C05471=1216.995,158.633,-53.196,-177.937,5.940,148.445
C05472=1217.000,158.384,-53.175,-177.940,5.938,148.445
C05473=1217.005,158.135,-53.154,-177.943,5.937,148.446
C05474=1217.009,157.886,-53.131,-177.945,5.936,148.446
C05475=1217.014,157.637,-53.110,-177.947,5.934,148.446
C05476=1217.019,157.388,-53.089,-177.950,5.933,148.447
C05477=1217.023,157.139,-53.067,-177.953,5.931,148.447
C05478=1217.028,156.890,-53.046,-177.955,5.930,148.448
C05479=1217.033,156.641,-53.025,-177.958,5.929,148.448
C05480=1217.038,156.393,-53.003,-177.961,5.927,148.449
C05481=1217.042,156.143,-52.982,-177.963,5.926,148.449
C05482=1217.047,155.894,-52.960,-177.966,5.925,148.450
C05483=1217.052,155.645,-52.938,-177.968,5.923,148.450
C05484=1217.056,155.396,-52.918,-177.971,5.922,148.451
C05485=1217.061,155.147,-52.896,-177.974,5.920,148.451
C05486=1217.066,154.898,-52.875,-177.976,5.919,148.452
C05487=1217.071,154.649,-52.853,-177.979,5.918,148.452
C05488=1217.075,154.400,-52.831,-177.981,5.917,148.452
C05489=1217.080,154.151,-52.810,-177.984,5.915,148.453
C05490=1217.084,153.902,-52.789,-177.986,5.913,148.453
C05491=1217.089,153.652,-52.768,-177.989,5.912,148.454
C05492=1217.094,153.404,-52.746,-177.992,5.911,148.454
C05493=1217.099,153.154,-52.725,-177.994,5.910,148.455
C05494=1217.104,152.906,-52.704,-177.996,5.908,148.455
C05495=1217.108,152.657,-52.683,-177.999,5.907,148.456
C05496=1217.113,152.407,-52.661,-178.002,5.906,148.456
C05497=1217.118,152.158,-52.640,-178.004,5.905,148.456
C05498=1217.123,151.909,-52.618,-178.007,5.903,148.457
C05499=1217.127,151.661,-52.598,-178.010,5.901,148.457
C05500=1217.131,151.411,-52.576,-178.012,5.900,148.458
C05501=1217.137,151.162,-52.555,-178.015,5.899,148.458
C05502=1217.141,150.913,-52.535,-178.017,5.898,148.459
C05503=1217.146,150.664,-52.513,-178.020,5.896,148.459
C05504=1217.151,150.415,-52.492,-178.022,5.896,148.460
C05505=1217.155,150.166,-52.470,-178.025,5.894,148.460
C05506=1217.160,149.917,-52.450,-178.027,5.893,148.461
C05507=1217.165,149.668,-52.429,-178.030,5.891,148.461
C05508=1217.170,149.419,-52.407,-178.033,5.889,148.462
C05509=1217.174,149.170,-52.387,-178.036,5.889,148.462
C05510=1217.178,148.921,-52.365,-178.038,5.887,148.463
C05511=1217.184,148.671,-52.344,-178.040,5.886,148.463
C05512=1217.188,148.422,-52.323,-178.043,5.885,148.464
C05513=1217.193,148.173,-52.302,-178.046,5.884,148.464
C05514=1217.198,147.925,-52.281,-178.048,5.882,148.464
C05515=1217.203,147.676,-52.260,-178.051,5.881,148.465
C05516=1217.207,147.426,-52.239,-178.053,5.879,148.465
C05517=1217.211,147.177,-52.218,-178.056,5.878,148.466
C05518=1217.216,146.928,-52.197,-178.059,5.877,148.466
C05519=1217.222,146.679,-52.176,-178.061,5.876,148.467
C05520=1217.226,146.430,-52.155,-178.064,5.874,148.467
C05521=1217.231,146.181,-52.134,-178.066,5.874,148.468
C05522=1217.235,145.932,-52.113,-178.069,5.872,148.468
C05523=1217.240,145.682,-52.092,-178.071,5.871,148.469
C05524=1217.245,145.433,-52.071,-178.074,5.869,148.469
C05525=1217.249,145.185,-52.050,-178.076,5.868,148.470
C05526=1217.254,144.935,-52.029,-178.079,5.867,148.470
C05527=1217.259,144.686,-52.009,-178.082,5.865,148.470
C05528=1217.264,144.437,-51.988,-178.084,5.864,148.471
C05529=1217.268,144.188,-51.967,-178.087,5.863,148.471
C05530=1217.274,143.939,-51.946,-178.089,5.862,148.472
C05531=1217.278,143.691,-51.925,-178.093,5.860,148.472
C05532=1217.283,143.441,-51.904,-178.095,5.859,148.473
C05533=1217.287,143.192,-51.884,-178.097,5.857,148.473
C05534=1217.292,142.942,-51.863,-178.100,5.857,148.474
C05535=1217.296,142.694,-51.842,-178.103,5.855,148.474
C05536=1217.302,142.444,-51.821,-178.105,5.854,148.475
C05537=1217.306,142.195,-51.801,-178.108,5.853,148.475
C05538=1217.311,141.946,-51.780,-178.110,5.852,148.476
C05539=1217.316,141.697,-51.760,-178.113,5.850,148.476
C05540=1217.321,141.448,-51.739,-178.115,5.849,148.477
C05541=1217.325,141.199,-51.718,-178.118,5.848,148.477
C05542=1217.330,140.950,-51.697,-178.121,5.847,148.478
C05543=1217.335,140.701,-51.677,-178.123,5.846,148.478
C05544=1217.339,140.452,-51.657,-178.126,5.844,148.479
C05545=1217.344,140.202,-51.636,-178.128,5.843,148.479
C05546=1217.349,139.954,-51.615,-178.131,5.842,148.480
C05547=1217.354,139.704,-51.594,-178.133,5.841,148.480
C05548=1217.359,139.455,-51.574,-178.136,5.839,148.480
C05549=1217.364,139.206,-51.553,-178.138,5.838,148.481
C05550=1217.368,138.957,-51.533,-178.141,5.837,148.482
C05551=1217.373,138.708,-51.512,-178.144,5.836,148.482
C05552=1217.378,138.459,-51.491,-178.146,5.834,148.483
C05553=1217.382,138.210,-51.471,-178.149,5.833,148.483
C05554=1217.387,137.961,-51.450,-178.152,5.832,148.484
C05555=1217.392,137.712,-51.429,-178.154,5.831,148.484
C05556=1217.396,137.463,-51.409,-178.157,5.829,148.485
C05557=1217.401,137.214,-51.388,-178.159,5.828,148.485
C05558=1217.406,136.965,-51.368,-178.162,5.827,148.486
C05559=1217.410,136.716,-51.347,-178.164,5.826,148.486
C05560=1217.416,136.466,-51.327,-178.167,5.824,148.486
C05561=1217.420,136.217,-51.307,-178.170,5.824,148.487
C05562=1217.425,135.968,-51.286,-178.172,5.823,148.487
C05563=1217.429,135.719,-51.266,-178.175,5.821,148.488
C05564=1217.434,135.470,-51.245,-178.177,5.820,148.488
C05565=1217.439,135.221,-51.225,-178.180,5.819,148.489
C05566=1217.443,134.971,-51.205,-178.182,5.818,148.489
C05567=1217.449,134.722,-51.184,-178.185,5.816,148.490
C05568=1217.453,134.473,-51.164,-178.188,5.815,148.490
C05569=1217.457,134.224,-51.143,-178.190,5.814,148.491
C05570=1217.462,133.974,-51.124,-178.193,5.813,148.491
C05571=1217.468,133.706,-51.101,-178.196,5.811,148.492
C05572=1217.473,133.437,-51.080,-178.198,5.810,148.492
C05573=1217.478,133.169,-51.058,-178.201,5.809,148.493
C05574=1217.483,132.900,-51.036,-178.204,5.807,148.493
C05575=1217.488,132.651,-51.016,-178.207,5.807,148.494
C05576=1217.492,132.402,-50.995,-178.209,5.806,148.494
C05577=1217.498,132.153,-50.974,-178.212,5.804,148.495
C05578=1217.502,131.903,-50.955,-178.214,5.803,148.495
C05579=1217.507,131.654,-50.934,-178.217,5.801,148.496
C05580=1217.511,131.406,-50.914,-178.219,5.801,148.497
C05581=1217.517,131.156,-50.894,-178.222,5.799,148.497
C05582=1217.522,130.907,-50.874,-178.225,5.798,148.498
C05583=1217.526,130.658,-50.854,-178.227,5.797,148.498
C05584=1217.531,130.409,-50.834,-178.230,5.796,148.499
C05585=1217.535,130.160,-50.813,-178.232,5.795,148.499
C05586=1217.540,129.910,-50.794,-178.235,5.794,148.500
C05587=1217.545,129.661,-50.773,-178.237,5.793,148.500
C05588=1217.550,129.412,-50.753,-178.240,5.791,148.501
C05589=1217.555,129.163,-50.733,-178.243,5.790,148.501
C05590=1217.559,128.914,-50.713,-178.245,5.790,148.502
C05591=1217.564,128.665,-50.693,-178.248,5.788,148.502
C05592=1217.569,128.416,-50.673,-178.250,5.787,148.503
C05593=1217.573,128.166,-50.653,-178.253,5.785,148.503
C05594=1217.578,127.917,-50.633,-178.255,5.784,148.503
C05595=1217.583,127.668,-50.613,-178.258,5.783,148.504
C05596=1217.588,127.419,-50.592,-178.260,5.782,148.504
C05597=1217.593,127.170,-50.573,-178.263,5.781,148.505
C05598=1217.597,126.921,-50.552,-178.266,5.780,148.505
C05599=1217.602,126.671,-50.533,-178.268,5.779,148.506
C05600=1217.607,126.423,-50.513,-178.271,5.777,148.507
C05601=1217.612,126.173,-50.493,-178.274,5.777,148.507
C05602=1217.616,125.924,-50.473,-178.276,5.776,148.508
C05603=1217.621,125.675,-50.453,-178.279,5.774,148.508
C05604=1217.626,125.426,-50.433,-178.281,5.773,148.509
C05605=1217.631,125.177,-50.413,-178.284,5.772,148.509
C05606=1217.636,124.927,-50.394,-178.286,5.771,148.510
C05607=1217.640,124.678,-50.373,-178.289,5.770,148.510
C05608=1217.645,124.429,-50.354,-178.292,5.768,148.511
C05609=1217.649,124.180,-50.333,-178.294,5.768,148.511
C05610=1217.655,123.931,-50.314,-178.296,5.767,148.512
C05611=1217.659,123.681,-50.294,-178.300,5.765,148.512
C05612=1217.664,123.433,-50.274,-178.302,5.764,148.513
C05613=1217.669,123.183,-50.254,-178.305,5.763,148.513
C05614=1217.674,122.934,-50.235,-178.307,5.762,148.514
C05615=1217.678,122.685,-50.215,-178.310,5.761,148.514
C05616=1217.683,122.436,-50.195,-178.312,5.760,148.515
C05617=1217.688,122.187,-50.176,-178.315,5.759,148.515
C05618=1217.693,121.938,-50.155,-178.317,5.758,148.516
C05619=1217.698,121.688,-50.136,-178.320,5.757,148.516
C05620=1217.702,121.439,-50.116,-178.322,5.756,148.517
C05621=1217.708,121.190,-50.097,-178.325,5.754,148.517
C05622=1217.712,120.941,-50.076,-178.328,5.753,148.518
C05623=1217.716,120.692,-50.057,-178.330,5.753,148.519
C05624=1217.722,120.443,-50.038,-178.333,5.751,148.519
C05625=1217.726,120.193,-50.018,-178.335,5.750,148.520
C05626=1217.731,119.944,-49.998,-178.338,5.749,148.520
C05627=1217.735,119.695,-49.978,-178.341,5.748,148.521
C05628=1217.741,119.446,-49.959,-178.343,5.747,148.521
C05629=1217.746,119.196,-49.939,-178.346,5.745,148.522
C05630=1217.750,118.947,-49.920,-178.348,5.744,148.522
C05631=1217.755,118.698,-49.900,-178.351,5.744,148.523
C05632=1217.759,118.449,-49.881,-178.353,5.742,148.523
C05633=1217.764,118.199,-49.861,-178.356,5.741,148.524
C05634=1217.769,117.951,-49.842,-178.359,5.741,148.524
C05635=1217.774,117.701,-49.822,-178.361,5.739,148.525
C05636=1217.779,117.451,-49.802,-178.364,5.738,148.525
C05637=1217.784,117.203,-49.783,-178.366,5.737,148.526
C05638=1217.788,116.954,-49.763,-178.369,5.736,148.526
C05639=1217.793,116.705,-49.744,-178.371,5.735,148.527
C05640=1217.798,116.456,-49.724,-178.374,5.734,148.527
C05641=1217.803,116.206,-49.705,-178.377,5.733,148.528
C05642=1217.808,115.957,-49.685,-178.379,5.732,148.528
C05643=1217.812,115.708,-49.666,-178.381,5.731,148.529
C05644=1217.817,115.458,-49.647,-178.385,5.730,148.530
C05645=1217.822,115.209,-49.627,-178.387,5.729,148.530
C05646=1217.827,114.960,-49.608,-178.389,5.728,148.531
C05647=1217.832,114.711,-49.588,-178.393,5.727,148.531
C05648=1217.836,114.462,-49.569,-178.395,5.726,148.532
C05649=1217.841,114.212,-49.550,-178.397,5.725,148.532
C05650=1217.846,113.963,-49.530,-178.400,5.723,148.533
C05651=1217.851,113.714,-49.511,-178.403,5.723,148.533
C05652=1217.856,113.465,-49.492,-178.405,5.722,148.534
C05653=1217.860,113.216,-49.472,-178.408,5.720,148.534
C05654=1217.866,112.967,-49.453,-178.410,5.719,148.535
C05655=1217.870,112.717,-49.434,-178.413,5.719,148.535
C05656=1217.875,112.468,-49.414,-178.415,5.717,148.536
C05657=1217.880,112.219,-49.395,-178.418,5.716,148.536
C05658=1217.885,111.969,-49.375,-178.420,5.716,148.537
C05659=1217.889,111.721,-49.357,-178.423,5.714,148.537
C05660=1217.894,111.471,-49.337,-178.426,5.713,148.538
C05661=1217.899,111.222,-49.318,-178.428,5.712,148.539
C05662=1217.904,110.973,-49.299,-178.431,5.712,148.539
C05663=1217.909,110.724,-49.280,-178.433,5.710,148.540
C05664=1217.914,110.474,-49.261,-178.436,5.709,148.540
C05665=1217.918,110.225,-49.241,-178.438,5.709,148.541
C05666=1217.923,109.976,-49.222,-178.441,5.707,148.541
C05667=1217.927,109.727,-49.203,-178.444,5.706,148.542
C05668=1217.932,109.478,-49.184,-178.446,5.705,148.542
C05669=1217.937,109.228,-49.165,-178.449,5.704,148.543
C05670=1217.942,108.979,-49.146,-178.451,5.703,148.543
C05671=1217.947,108.730,-49.127,-178.454,5.702,148.544
C05672=1217.952,108.481,-49.107,-178.457,5.701,148.545
C05673=1217.956,108.231,-49.088,-178.459,5.700,148.545
C05674=1217.962,107.982,-49.070,-178.462,5.699,148.546
C05675=1217.966,107.714,-49.049,-178.464,5.698,148.546
C05676=1217.972,107.446,-49.028,-178.467,5.697,148.547
C05677=1217.977,107.176,-49.008,-178.470,5.696,148.547
C05678=1217.982,106.909,-48.987,-178.473,5.695,148.548
C05679=1217.986,106.659,-48.968,-178.475,5.694,148.548
C05680=1217.992,106.410,-48.950,-178.478,5.693,148.549
C05681=1217.997,106.161,-48.931,-178.481,5.692,148.550
C05682=1218.001,105.912,-48.911,-178.483,5.691,148.550
C05683=1218.007,105.662,-48.893,-178.485,5.690,148.551
C05684=1218.011,105.413,-48.874,-178.488,5.689,148.551
C05685=1218.016,105.164,-48.854,-178.491,5.688,148.552
C05686=1218.021,104.914,-48.836,-178.493,5.687,148.552
C05687=1218.026,104.665,-48.817,-178.496,5.687,148.553
C05688=1218.030,104.416,-48.798,-178.499,5.685,148.553
C05689=1218.036,104.167,-48.779,-178.501,5.684,148.554
C05690=1218.040,103.918,-48.760,-178.503,5.684,148.555
C05691=1218.045,103.668,-48.741,-178.507,5.682,148.555
C05692=1218.050,103.419,-48.723,-178.509,5.681,148.556
C05693=1218.054,103.170,-48.704,-178.511,5.681,148.556
C05694=1218.059,102.920,-48.685,-178.513,5.680,148.557
C05695=1218.063,102.671,-48.666,-178.517,5.678,148.557
C05696=1218.069,102.422,-48.648,-178.519,5.678,148.558
C05697=1218.074,102.173,-48.629,-178.521,5.677,148.558
C05698=1218.078,101.924,-48.609,-178.524,5.676,148.559
C05699=1218.083,101.674,-48.591,-178.527,5.674,148.559
C05700=1218.088,101.425,-48.572,-178.529,5.674,148.560
C05701=1218.093,101.176,-48.554,-178.532,5.673,148.561
C05702=1218.098,100.927,-48.535,-178.534,5.672,148.561
C05703=1218.103,100.677,-48.516,-178.537,5.671,148.562
C05704=1218.107,100.428,-48.497,-178.540,5.670,148.562
C05705=1218.113,100.179,-48.479,-178.542,5.669,148.563
C05706=1218.117,99.930,-48.460,-178.545,5.669,148.563
C05707=1218.122,99.680,-48.442,-178.547,5.667,148.564
C05708=1218.127,99.431,-48.422,-178.550,5.666,148.565
C05709=1218.132,99.182,-48.404,-178.553,5.666,148.565
C05710=1218.136,98.933,-48.385,-178.555,5.665,148.566
C05711=1218.141,98.683,-48.366,-178.558,5.663,148.566
C05712=1218.146,98.434,-48.348,-178.560,5.662,148.567
C05713=1218.151,98.185,-48.330,-178.563,5.662,148.567
C05714=1218.156,97.935,-48.311,-178.565,5.661,148.568
C05715=1218.160,97.687,-48.292,-178.568,5.659,148.568
C05716=1218.165,97.437,-48.274,-178.571,5.659,148.569
C05717=1218.170,97.187,-48.255,-178.573,5.658,148.570
C05718=1218.175,96.939,-48.236,-178.575,5.657,148.570
C05719=1218.180,96.689,-48.218,-178.578,5.656,148.571
C05720=1218.185,96.440,-48.200,-178.581,5.655,148.571
C05721=1218.190,96.191,-48.181,-178.583,5.654,148.572
C05722=1218.194,95.942,-48.163,-178.586,5.654,148.572
C05723=1218.199,95.692,-48.145,-178.588,5.653,148.573
C05724=1218.204,95.443,-48.125,-178.591,5.651,148.573
C05725=1218.209,95.194,-48.107,-178.594,5.651,148.574
C05726=1218.214,94.944,-48.089,-178.596,5.650,148.575
C05727=1218.219,94.695,-48.070,-178.599,5.649,148.575
C05728=1218.224,94.446,-48.052,-178.602,5.648,148.576
C05729=1218.228,94.196,-48.034,-178.604,5.647,148.576
C05730=1218.233,93.947,-48.016,-178.606,5.646,148.577
C05731=1218.237,93.698,-47.997,-178.609,5.646,148.578
C05732=1218.243,93.449,-47.978,-178.611,5.645,148.578
C05733=1218.248,93.199,-47.960,-178.614,5.643,148.579
C05734=1218.253,92.950,-47.942,-178.617,5.643,148.579
C05735=1218.257,92.701,-47.923,-178.619,5.642,148.580
C05736=1218.262,92.452,-47.905,-178.622,5.641,148.580
C05737=1218.267,92.202,-47.886,-178.624,5.640,148.581
C05738=1218.272,91.953,-47.868,-178.627,5.639,148.581
C05739=1218.277,91.703,-47.850,-178.630,5.638,148.582
C05740=1218.281,91.455,-47.831,-178.632,5.638,148.583
C05741=1218.286,91.206,-47.813,-178.634,5.637,148.583
C05742=1218.291,90.956,-47.795,-178.637,5.636,148.584
C05743=1218.297,90.707,-47.777,-178.640,5.635,148.584
C05744=1218.301,90.457,-47.759,-178.642,5.634,148.585
C05745=1218.306,90.208,-47.741,-178.645,5.633,148.585
C05746=1218.311,89.959,-47.723,-178.648,5.632,148.586
C05747=1218.316,89.709,-47.705,-178.650,5.632,148.587
C05748=1218.320,89.461,-47.686,-178.653,5.630,148.587
C05749=1218.325,89.211,-47.668,-178.656,5.630,148.588
C05750=1218.330,88.962,-47.649,-178.658,5.629,148.588
C05751=1218.335,88.712,-47.631,-178.660,5.628,148.589
C05752=1218.340,88.463,-47.613,-178.663,5.627,148.590
C05753=1218.345,88.214,-47.595,-178.665,5.626,148.590
C05754=1218.349,87.964,-47.577,-178.668,5.625,148.591
C05755=1218.354,87.715,-47.559,-178.671,5.624,148.591
C05756=1218.359,87.466,-47.541,-178.673,5.624,148.592
C05757=1218.364,87.217,-47.523,-178.676,5.623,148.592
C05758=1218.369,86.967,-47.505,-178.678,5.622,148.593
C05759=1218.374,86.718,-47.487,-178.681,5.621,148.593
C05760=1218.378,86.468,-47.468,-178.684,5.620,148.594
C05761=1218.383,86.219,-47.450,-178.686,5.619,148.595
C05762=1218.388,85.970,-47.432,-178.688,5.618,148.595
C05763=1218.393,85.721,-47.414,-178.691,5.618,148.596
C05764=1218.398,85.472,-47.396,-178.694,5.617,148.596
C05765=1218.403,85.222,-47.379,-178.696,5.616,148.597
C05766=1218.408,84.973,-47.361,-178.699,5.615,148.598
C05767=1218.413,84.724,-47.343,-178.702,5.614,148.598
C05768=1218.417,84.474,-47.324,-178.704,5.614,148.599
C05769=1218.422,84.225,-47.306,-178.706,5.613,148.599
C05770=1218.427,83.975,-47.289,-178.709,5.612,148.600
C05771=1218.432,83.726,-47.271,-178.712,5.611,148.601
C05772=1218.437,83.477,-47.253,-178.714,5.610,148.601
C05773=1218.442,83.228,-47.235,-178.717,5.609,148.602
C05774=1218.447,82.979,-47.217,-178.720,5.609,148.602
C05775=1218.452,82.729,-47.199,-178.722,5.608,148.603
C05776=1218.457,82.480,-47.181,-178.724,5.607,148.603
C05777=1218.462,82.230,-47.164,-178.727,5.607,148.604
C05778=1218.466,81.981,-47.145,-178.730,5.605,148.605
C05779=1218.472,81.713,-47.126,-178.732,5.604,148.605
C05780=1218.477,81.445,-47.107,-178.735,5.604,148.606
C05781=1218.482,81.176,-47.088,-178.738,5.602,148.606
C05782=1218.487,80.908,-47.069,-178.741,5.602,148.607
C05783=1218.492,80.658,-47.051,-178.743,5.601,148.608
C05784=1218.497,80.409,-47.033,-178.746,5.601,148.608
C05785=1218.502,80.159,-47.016,-178.748,5.600,148.609
C05786=1218.507,79.910,-46.998,-178.751,5.599,148.609
C05787=1218.512,79.661,-46.980,-178.754,5.598,148.610
C05788=1218.516,79.412,-46.962,-178.756,5.597,148.611
C05789=1218.522,79.162,-46.945,-178.759,5.596,148.611
C05790=1218.526,78.913,-46.927,-178.761,5.596,148.612
C05791=1218.531,78.664,-46.909,-178.764,5.595,148.613
C05792=1218.536,78.414,-46.891,-178.766,5.594,148.613
C05793=1218.541,78.164,-46.874,-178.769,5.593,148.614
C05794=1218.546,77.915,-46.856,-178.771,5.593,148.614
C05795=1218.550,77.666,-46.838,-178.774,5.591,148.615
C05796=1218.555,77.417,-46.821,-178.777,5.591,148.615
C05797=1218.560,77.167,-46.803,-178.779,5.590,148.616
C05798=1218.565,76.918,-46.785,-178.782,5.589,148.617
C05799=1218.570,76.668,-46.768,-178.784,5.588,148.617
C05800=1218.574,76.420,-46.750,-178.787,5.588,148.618
C05801=1218.580,76.170,-46.733,-178.789,5.587,148.618
C05802=1218.585,75.921,-46.715,-178.792,5.587,148.619
C05803=1218.590,75.672,-46.697,-178.795,5.585,148.619
C05804=1218.595,75.422,-46.680,-178.797,5.584,148.620
C05805=1218.599,75.174,-46.663,-178.800,5.584,148.621
C05806=1218.605,74.924,-46.646,-178.802,5.583,148.621
C05807=1218.610,74.675,-46.628,-178.805,5.582,148.622
C05808=1218.615,74.425,-46.610,-178.807,5.582,148.623
C05809=1218.619,74.176,-46.593,-178.810,5.581,148.623
C05810=1218.624,73.927,-46.575,-178.812,5.580,148.624
C05811=1218.629,73.677,-46.558,-178.815,5.580,148.624
C05812=1218.633,73.428,-46.540,-178.818,5.578,148.625
C05813=1218.639,73.178,-46.523,-178.820,5.578,148.626
C05814=1218.643,72.929,-46.505,-178.823,5.577,148.626
C05815=1218.649,72.679,-46.488,-178.825,5.576,148.627
C05816=1218.653,72.430,-46.470,-178.828,5.576,148.627
C05817=1218.658,72.181,-46.453,-178.830,5.575,148.628
C05818=1218.663,71.931,-46.435,-178.833,5.574,148.628
C05819=1218.667,71.682,-46.418,-178.835,5.573,148.629
C05820=1218.673,71.433,-46.401,-178.838,5.573,148.630
C05821=1218.678,71.184,-46.384,-178.841,5.572,148.630
C05822=1218.683,70.934,-46.367,-178.843,5.571,148.631
C05823=1218.688,70.685,-46.349,-178.846,5.570,148.632
C05824=1218.693,70.435,-46.332,-178.848,5.569,148.632
C05825=1218.697,70.186,-46.314,-178.851,5.569,148.633
C05826=1218.702,69.937,-46.297,-178.853,5.568,148.633
C05827=1218.707,69.687,-46.279,-178.856,5.567,148.634
C05828=1218.712,69.438,-46.262,-178.859,5.567,148.635
C05829=1218.717,69.188,-46.245,-178.861,5.566,148.635
C05830=1218.722,68.940,-46.228,-178.863,5.565,148.636
C05831=1218.727,68.690,-46.211,-178.866,5.565,148.636
C05832=1218.732,68.440,-46.194,-178.869,5.564,148.637
C05833=1218.736,68.191,-46.176,-178.871,5.564,148.638
C05834=1218.741,67.942,-46.159,-178.874,5.562,148.638
C05835=1218.746,67.692,-46.142,-178.877,5.561,148.639
C05836=1218.751,67.443,-46.124,-178.879,5.561,148.639
C05837=1218.757,67.194,-46.107,-178.882,5.560,148.640
C05838=1218.761,66.944,-46.091,-178.884,5.560,148.641
C05839=1218.766,66.695,-46.073,-178.887,5.559,148.641
C05840=1218.770,66.446,-46.056,-178.889,5.558,148.642
C05841=1218.776,66.196,-46.039,-178.892,5.557,148.643
C05842=1218.780,65.947,-46.022,-178.894,5.557,148.643
C05843=1218.786,65.698,-46.004,-178.897,5.556,148.644
C05844=1218.790,65.449,-45.988,-178.899,5.555,148.644
C05845=1218.795,65.199,-45.971,-178.902,5.555,148.645
C05846=1218.800,64.949,-45.954,-178.904,5.554,148.646
C05847=1218.805,64.700,-45.936,-178.907,5.554,148.646
C05848=1218.810,64.451,-45.920,-178.909,5.553,148.647
C05849=1218.815,64.202,-45.902,-178.912,5.551,148.647
C05850=1218.820,63.952,-45.886,-178.915,5.551,148.648
C05851=1218.825,63.702,-45.868,-178.918,5.550,148.649
C05852=1218.829,63.453,-45.851,-178.920,5.549,148.649
C05853=1218.835,63.204,-45.834,-178.922,5.549,148.650
C05854=1218.839,62.955,-45.817,-178.925,5.548,148.650
C05855=1218.844,62.705,-45.800,-178.928,5.548,148.651
C05856=1218.849,62.456,-45.784,-178.930,5.547,148.652
C05857=1218.855,62.206,-45.767,-178.933,5.546,148.652
C05858=1218.859,61.958,-45.749,-178.935,5.546,148.653
C05859=1218.864,61.708,-45.732,-178.938,5.545,148.654
C05860=1218.869,61.458,-45.715,-178.940,5.544,148.654
C05861=1218.873,61.209,-45.699,-178.943,5.543,148.655
C05862=1218.879,60.960,-45.682,-178.945,5.543,148.655
C05863=1218.883,60.710,-45.665,-178.948,5.542,148.656
C05864=1218.889,60.460,-45.648,-178.950,5.542,148.657
C05865=1218.894,60.212,-45.631,-178.953,5.541,148.657
C05866=1218.898,59.962,-45.615,-178.955,5.540,148.658
C05867=1218.903,59.712,-45.598,-178.958,5.540,148.658
C05868=1218.908,59.463,-45.581,-178.960,5.539,148.659
C05869=1218.914,59.214,-45.564,-178.963,5.539,148.660
C05870=1218.918,58.964,-45.547,-178.966,5.538,148.660
C05871=1218.923,58.715,-45.531,-178.968,5.537,148.661
C05872=1218.928,58.466,-45.514,-178.971,5.537,148.661
C05873=1218.933,58.216,-45.497,-178.974,5.535,148.662
C05874=1218.937,57.967,-45.480,-178.976,5.535,148.663
C05875=1218.943,57.717,-45.463,-178.979,5.534,148.663
C05876=1218.948,57.468,-45.447,-178.981,5.533,148.664
C05877=1218.952,57.219,-45.430,-178.984,5.533,148.665
C05878=1218.957,56.969,-45.413,-178.986,5.532,148.665
C05879=1218.963,56.720,-45.397,-178.989,5.531,148.666
C05880=1218.967,56.471,-45.380,-178.992,5.531,148.667
C05881=1218.972,56.221,-45.363,-178.994,5.530,148.667
C05882=1218.977,55.972,-45.346,-178.996,5.529,148.668
C05883=1218.982,55.703,-45.328,-178.999,5.529,148.668
C05884=1218.988,55.435,-45.311,-179.002,5.528,148.669
C05885=1218.993,55.166,-45.293,-179.004,5.528,148.670
C05886=1218.998,54.898,-45.275,-179.007,5.527,148.670
C05887=1219.003,54.648,-45.258,-179.010,5.527,148.671
C05888=1219.008,54.400,-45.241,-179.012,5.526,148.672
C05889=1219.013,54.150,-45.225,-179.015,5.525,148.672
C05890=1219.018,53.900,-45.208,-179.018,5.525,148.673
C05891=1219.024,53.651,-45.192,-179.020,5.524,148.673
C05892=1219.028,53.402,-45.175,-179.022,5.523,148.674
C05893=1219.032,53.152,-45.158,-179.025,5.523,148.675
C05894=1219.038,52.903,-45.142,-179.028,5.522,148.675
C05895=1219.043,52.653,-45.125,-179.030,5.522,148.676
C05896=1219.048,52.404,-45.109,-179.033,5.521,148.677
C05897=1219.053,52.155,-45.093,-179.035,5.520,148.677
C05898=1219.057,51.905,-45.076,-179.038,5.520,148.678
C05899=1219.063,51.656,-45.059,-179.040,5.519,148.679
C05900=1219.068,51.406,-45.043,-179.043,5.519,148.679
C05901=1219.072,51.156,-45.026,-179.046,5.518,148.680
C05902=1219.077,50.908,-45.010,-179.048,5.517,148.680
C05903=1219.082,50.658,-44.993,-179.050,5.517,148.681
C05904=1219.087,50.409,-44.978,-179.053,5.516,148.682
C05905=1219.092,50.159,-44.961,-179.056,5.515,148.682
C05906=1219.097,49.910,-44.944,-179.058,5.515,148.683
C05907=1219.102,49.661,-44.928,-179.061,5.514,148.684
C05908=1219.107,49.411,-44.912,-179.063,5.513,148.684
C05909=1219.112,49.162,-44.895,-179.066,5.513,148.685
C05910=1219.116,48.912,-44.879,-179.068,5.512,148.685
C05911=1219.122,48.663,-44.863,-179.071,5.512,148.686
C05912=1219.127,48.413,-44.846,-179.074,5.511,148.687
C05913=1219.132,48.164,-44.830,-179.076,5.511,148.688
C05914=1219.137,47.914,-44.814,-179.078,5.510,148.688
C05915=1219.142,47.665,-44.797,-179.081,5.509,148.689
C05916=1219.146,47.416,-44.781,-179.084,5.509,148.689
C05917=1219.151,47.166,-44.765,-179.086,5.508,148.690
C05918=1219.156,46.917,-44.748,-179.089,5.507,148.691
C05919=1219.161,46.667,-44.732,-179.092,5.507,148.691
C05920=1219.166,46.418,-44.716,-179.094,5.506,148.692
C05921=1219.171,46.169,-44.699,-179.096,5.505,148.692
C05922=1219.176,45.919,-44.684,-179.099,5.505,148.693
C05923=1219.180,45.670,-44.667,-179.102,5.504,148.694
C05924=1219.187,45.420,-44.651,-179.104,5.504,148.694
C05925=1219.191,45.171,-44.634,-179.107,5.503,148.695
C05926=1219.196,44.921,-44.619,-179.110,5.503,148.696
C05927=1219.201,44.672,-44.602,-179.112,5.502,148.696
C05928=1219.206,44.422,-44.586,-179.114,5.501,148.697
C05929=1219.211,44.173,-44.570,-179.117,5.501,148.698
C05930=1219.216,43.924,-44.553,-179.120,5.500,148.698
C05931=1219.221,43.674,-44.538,-179.122,5.500,148.699
C05932=1219.226,43.425,-44.521,-179.125,5.499,148.700
C05933=1219.230,43.175,-44.505,-179.127,5.498,148.700
C05934=1219.236,42.926,-44.490,-179.129,5.498,148.701
C05935=1219.241,42.677,-44.473,-179.132,5.498,148.701
C05936=1219.246,42.427,-44.457,-179.134,5.497,148.702
C05937=1219.251,42.178,-44.441,-179.137,5.497,148.703
C05938=1219.256,41.928,-44.425,-179.140,5.496,148.703
C05939=1219.261,41.679,-44.409,-179.142,5.496,148.704
C05940=1219.265,41.429,-44.393,-179.144,5.495,148.705
C05941=1219.271,41.180,-44.377,-179.147,5.494,148.705
C05942=1219.275,40.930,-44.361,-179.150,5.494,148.706
C05943=1219.280,40.681,-44.346,-179.152,5.493,148.707
C05944=1219.285,40.432,-44.329,-179.155,5.492,148.707
C05945=1219.290,40.182,-44.313,-179.158,5.492,148.708
C05946=1219.295,39.933,-44.297,-179.160,5.491,148.709
C05947=1219.300,39.683,-44.281,-179.162,5.490,148.709
C05948=1219.305,39.434,-44.266,-179.165,5.490,148.710
C05949=1219.310,39.184,-44.249,-179.168,5.489,148.710
C05950=1219.315,38.935,-44.233,-179.170,5.489,148.711
C05951=1219.320,38.686,-44.218,-179.173,5.488,148.712
C05952=1219.325,38.436,-44.201,-179.175,5.489,148.712
C05953=1219.330,38.187,-44.185,-179.178,5.488,148.713
C05954=1219.334,37.937,-44.170,-179.180,5.487,148.714
C05955=1219.339,37.688,-44.154,-179.182,5.487,148.714
C05956=1219.345,37.439,-44.138,-179.185,5.486,148.715
C05957=1219.350,37.189,-44.122,-179.188,5.485,148.716
C05958=1219.355,36.939,-44.107,-179.190,5.485,148.716
C05959=1219.360,36.690,-44.090,-179.193,5.484,148.717
C05960=1219.365,36.440,-44.074,-179.196,5.484,148.718
C05961=1219.370,36.191,-44.059,-179.198,5.483,148.718
C05962=1219.374,35.942,-44.043,-179.200,5.482,148.719
C05963=1219.379,35.692,-44.027,-179.203,5.482,148.719
C05964=1219.385,35.443,-44.012,-179.206,5.481,148.720
C05965=1219.389,35.193,-43.996,-179.208,5.482,148.721
C05966=1219.395,34.943,-43.980,-179.210,5.481,148.721
C05967=1219.399,34.695,-43.964,-179.213,5.480,148.722
C05968=1219.404,34.445,-43.948,-179.216,5.480,148.723
C05969=1219.409,34.195,-43.933,-179.218,5.479,148.723
C05970=1219.415,33.946,-43.917,-179.221,5.479,148.724
C05971=1219.420,33.696,-43.901,-179.223,5.478,148.725
C05972=1219.424,33.447,-43.886,-179.226,5.477,148.725
C05973=1219.429,33.198,-43.870,-179.228,5.477,148.726
C05974=1219.434,32.948,-43.854,-179.231,5.476,148.727
C05975=1219.439,32.699,-43.838,-179.234,5.476,148.727
C05976=1219.444,32.449,-43.823,-179.236,5.475,148.728
C05977=1219.449,32.199,-43.807,-179.238,5.475,148.729
C05978=1219.454,31.950,-43.792,-179.241,5.475,148.729
C05979=1219.460,31.701,-43.776,-179.243,5.474,148.730
C05980=1219.464,31.452,-43.761,-179.246,5.473,148.730
C05981=1219.469,31.202,-43.745,-179.249,5.473,148.731
C05982=1219.474,30.953,-43.729,-179.251,5.472,148.732
C05983=1219.479,30.704,-43.714,-179.254,5.472,148.732
C05984=1219.484,30.453,-43.698,-179.256,5.471,148.733
C05985=1219.489,30.204,-43.682,-179.259,5.471,148.734
C05986=1219.494,29.955,-43.667,-179.262,5.470,148.734
C05987=1219.499,29.686,-43.650,-179.264,5.470,148.735
C05988=1219.505,29.417,-43.634,-179.267,5.469,148.736
C05989=1219.510,29.148,-43.617,-179.270,5.469,148.736
C05990=1219.515,28.880,-43.600,-179.272,5.468,148.737
C05991=1219.520,28.631,-43.585,-179.275,5.468,148.738
C05992=1219.526,28.381,-43.569,-179.277,5.468,148.739
C05993=1219.530,28.132,-43.554,-179.280,5.467,148.739
C05994=1219.535,27.882,-43.538,-179.282,5.467,148.740
C05995=1219.540,27.633,-43.523,-179.285,5.466,148.741
C05996=1219.545,27.383,-43.508,-179.287,5.465,148.741
C05997=1219.550,27.134,-43.492,-179.290,5.465,148.742
C05998=1219.555,26.884,-43.476,-179.292,5.464,148.742
C05999=1219.560,26.635,-43.461,-179.295,5.464,148.743
C06000=1219.565,26.385,-43.446,-179.298,5.463,148.744
C06001=1219.570,26.136,-43.431,-179.300,5.463,148.744
C06002=1219.576,25.886,-43.416,-179.302,5.463,148.745
C06003=1219.580,25.636,-43.400,-179.305,5.462,148.746
C06004=1219.585,25.387,-43.385,-179.308,5.462,148.746
C06005=1219.590,25.138,-43.369,-179.310,5.461,148.747
C06006=1219.595,24.889,-43.354,-179.313,5.460,148.748
C06007=1219.600,24.639,-43.339,-179.315,5.460,148.748
C06008=1219.605,24.389,-43.323,-179.318,5.459,148.749
C06009=1219.610,24.140,-43.308,-179.320,5.460,148.750
C06010=1219.616,23.890,-43.293,-179.323,5.459,148.750
C06011=1219.620,23.641,-43.278,-179.325,5.458,148.751
C06012=1219.626,23.392,-43.262,-179.328,5.458,148.752
C06013=1219.630,23.142,-43.247,-179.330,5.457,148.752
C06014=1219.635,22.892,-43.231,-179.333,5.457,148.753
C06015=1219.640,22.643,-43.216,-179.336,5.456,148.754
C06016=1219.645,22.393,-43.201,-179.338,5.457,148.754
C06017=1219.650,22.144,-43.186,-179.340,5.456,148.755
C06018=1219.655,21.895,-43.171,-179.343,5.455,148.755
C06019=1219.660,21.646,-43.156,-179.345,5.455,148.756
C06020=1219.665,21.396,-43.140,-179.348,5.454,148.757
C06021=1219.670,21.146,-43.126,-179.351,5.454,148.758
C06022=1219.675,20.896,-43.110,-179.353,5.453,148.758
C06023=1219.680,20.647,-43.095,-179.355,5.453,148.759
C06024=1219.685,20.398,-43.079,-179.358,5.453,148.760
C06025=1219.690,20.148,-43.065,-179.361,5.452,148.760
C06026=1219.696,19.899,-43.050,-179.363,5.452,148.761
C06027=1219.700,19.650,-43.035,-179.366,5.451,148.762
C06028=1219.705,19.399,-43.019,-179.368,5.450,148.762
C06029=1219.710,19.150,-43.004,-179.371,5.450,148.763
C06030=1219.715,18.901,-42.989,-179.373,5.450,148.763
C06031=1219.720,18.651,-42.974,-179.375,5.450,148.764
C06032=1219.725,18.402,-42.959,-179.378,5.449,148.765
C06033=1219.730,18.152,-42.944,-179.381,5.448,148.765
C06034=1219.735,17.903,-42.929,-179.383,5.448,148.766
C06035=1219.741,17.653,-42.914,-179.386,5.447,148.767
C06036=1219.745,17.404,-42.899,-179.388,5.448,148.768
C06037=1219.750,17.154,-42.885,-179.391,5.447,148.768
C06038=1219.755,16.904,-42.869,-179.393,5.447,148.769
C06039=1219.760,16.655,-42.854,-179.396,5.446,148.770
C06040=1219.765,16.405,-42.839,-179.399,5.446,148.770
C06041=1219.770,16.156,-42.824,-179.401,5.445,148.771
C06042=1219.775,15.907,-42.809,-179.403,5.445,148.771
C06043=1219.780,15.657,-42.794,-179.406,5.444,148.772
C06044=1219.785,15.408,-42.779,-179.408,5.444,148.773
C06045=1219.790,15.158,-42.765,-179.411,5.443,148.773
C06046=1219.795,14.909,-42.749,-179.414,5.443,148.774
C06047=1219.800,14.659,-42.735,-179.416,5.442,148.775
C06048=1219.805,14.410,-42.720,-179.418,5.443,148.776
C06049=1219.811,14.160,-42.705,-179.421,5.442,148.776
C06050=1219.815,13.911,-42.690,-179.424,5.442,148.777
C06051=1219.820,13.662,-42.675,-179.426,5.441,148.778
C06052=1219.826,13.412,-42.660,-179.429,5.441,148.778
C06053=1219.830,13.163,-42.645,-179.431,5.440,148.779
C06054=1219.835,12.913,-42.631,-179.433,5.440,148.779
C06055=1219.841,12.664,-42.615,-179.436,5.439,148.780
C06056=1219.846,12.414,-42.601,-179.438,5.439,148.781
C06057=1219.851,12.164,-42.587,-179.441,5.438,148.781
C06058=1219.856,11.915,-42.571,-179.444,5.438,148.782
C06059=1219.861,11.665,-42.557,-179.446,5.437,148.783
C06060=1219.866,11.416,-42.542,-179.448,5.438,148.784
C06061=1219.871,11.166,-42.528,-179.451,5.437,148.784
C06062=1219.876,10.917,-42.512,-179.454,5.437,148.785
C06063=1219.881,10.667,-42.498,-179.456,5.436,148.786
C06064=1219.886,10.418,-42.483,-179.459,5.435,148.786
C06065=1219.891,10.168,-42.468,-179.461,5.436,148.787
C06066=1219.896,9.918,-42.454,-179.464,5.435,148.788
C06067=1219.901,9.669,-42.439,-179.466,5.435,148.788
C06068=1219.906,9.420,-42.424,-179.469,5.434,148.789
C06069=1219.910,9.170,-42.409,-179.471,5.433,148.789
C06070=1219.916,8.920,-42.394,-179.473,5.434,148.790
C06071=1219.921,8.671,-42.380,-179.476,5.433,148.791
C06072=1219.926,8.422,-42.365,-179.479,5.433,148.791
C06073=1219.931,8.172,-42.351,-179.481,5.432,148.792
C06074=1219.936,7.922,-42.337,-179.484,5.432,148.793
C06075=1219.941,7.673,-42.321,-179.486,5.432,148.794
C06076=1219.946,7.423,-42.307,-179.489,5.431,148.794
C06077=1219.951,7.173,-42.293,-179.491,5.431,148.795
C06078=1219.956,6.924,-42.278,-179.494,5.430,148.796
C06079=1219.961,6.675,-42.263,-179.497,5.430,148.796
C06080=1219.966,6.425,-42.249,-179.499,5.430,148.797
C06081=1219.971,6.176,-42.234,-179.501,5.429,148.798
C06082=1219.976,5.926,-42.219,-179.504,5.429,148.798
C06083=1219.981,5.677,-42.205,-179.507,5.428,148.799
C06084=1219.986,5.427,-42.191,-179.509,5.428,148.800
C06085=1219.991,5.178,-42.176,-179.511,5.428,148.800
C06086=1219.996,4.928,-42.162,-179.513,5.427,148.801
C06087=1220.001,4.678,-42.147,-179.516,5.427,148.802
C06088=1220.006,4.429,-42.133,-179.519,5.426,148.802
C06089=1220.011,4.179,-42.118,-179.521,5.426,148.803
C06090=1220.016,3.930,-42.103,-179.523,5.426,148.804
C06091=1220.022,3.661,-42.089,-179.526,5.426,148.804
C06092=1220.027,3.392,-42.073,-179.529,5.425,148.805
C06093=1220.033,3.123,-42.057,-179.532,5.425,148.806
C06094=1220.038,2.854,-42.042,-179.535,5.424,148.807
C06095=1220.043,2.605,-42.027,-179.537,5.424,148.807
C06096=1220.048,2.355,-42.013,-179.540,5.423,148.808
C06097=1220.053,2.105,-41.998,-179.542,5.424,148.809
C06098=1220.058,1.855,-41.984,-179.545,5.423,148.809
C06099=1220.064,1.606,-41.970,-179.547,5.423,148.810
C06100=1220.069,1.357,-41.956,-179.550,5.422,148.811
C06101=1220.073,1.108,-41.941,-179.552,5.422,148.811
C06102=1220.078,0.858,-41.926,-179.555,5.422,148.812
C06103=1220.083,0.608,-41.912,-179.557,5.421,148.813
C06104=1220.088,0.358,-41.898,-179.559,5.420,148.813
C06105=1220.094,0.109,-41.884,-179.562,5.420,148.814
C06106=1220.099,-0.140,-41.870,-179.564,5.420,148.815
C06107=1220.104,-0.390,-41.855,-179.567,5.420,148.815
C06108=1220.109,-0.640,-41.841,-179.569,5.419,148.816
C06109=1220.114,-0.889,-41.827,-179.572,5.419,148.817
C06110=1220.119,-1.139,-41.812,-179.574,5.419,148.817
C06111=1220.124,-1.388,-41.799,-179.577,5.418,148.818
C06112=1220.129,-1.638,-41.784,-179.580,5.418,148.819
C06113=1220.134,-1.888,-41.770,-179.582,5.417,148.819
C06114=1220.139,-2.137,-41.756,-179.584,5.418,148.820
C06115=1220.144,-2.387,-41.741,-179.587,5.417,148.821
C06116=1220.149,-2.636,-41.728,-179.590,5.417,148.822
C06117=1220.154,-2.886,-41.713,-179.592,5.416,148.822
C06118=1220.159,-3.135,-41.699,-179.595,5.416,148.823
C06119=1220.164,-3.385,-41.685,-179.597,5.416,148.824
C06120=1220.170,-3.634,-41.671,-179.600,5.415,148.824
C06121=1220.174,-3.883,-41.657,-179.602,5.415,148.825
C06122=1220.179,-4.133,-41.643,-179.605,5.414,148.826
C06123=1220.184,-4.383,-41.629,-179.607,5.415,148.826
C06124=1220.189,-4.633,-41.614,-179.610,5.414,148.827
C06125=1220.195,-4.882,-41.600,-179.612,5.413,148.828
C06126=1220.199,-5.131,-41.586,-179.614,5.413,148.828
C06127=1220.204,-5.381,-41.572,-179.617,5.413,148.829
C06128=1220.209,-5.631,-41.558,-179.619,5.413,148.830
C06129=1220.215,-5.880,-41.544,-179.622,5.412,148.830
C06130=1220.220,-6.129,-41.529,-179.624,5.412,148.831
C06131=1220.224,-6.379,-41.516,-179.627,5.412,148.832
C06132=1220.229,-6.629,-41.501,-179.629,5.411,148.832
C06133=1220.235,-6.878,-41.488,-179.632,5.411,148.833
C06134=1220.240,-7.128,-41.474,-179.635,5.410,148.834
C06135=1220.245,-7.378,-41.460,-179.637,5.411,148.834
C06136=1220.250,-7.627,-41.446,-179.639,5.410,148.835
C06137=1220.255,-7.876,-41.431,-179.642,5.410,148.836
C06138=1220.260,-8.126,-41.418,-179.644,5.410,148.837
C06139=1220.265,-8.375,-41.403,-179.647,5.409,148.837
C06140=1220.270,-8.625,-41.390,-179.649,5.409,148.838
C06141=1220.275,-8.875,-41.376,-179.652,5.408,148.839
C06142=1220.280,-9.125,-41.362,-179.654,5.409,148.839
C06143=1220.285,-9.373,-41.348,-179.657,5.408,148.840
C06144=1220.290,-9.623,-41.334,-179.659,5.408,148.841
C06145=1220.295,-9.873,-41.321,-179.662,5.407,148.841
C06146=1220.301,-10.122,-41.307,-179.664,5.408,148.842
C06147=1220.306,-10.372,-41.292,-179.667,5.407,148.843
C06148=1220.310,-10.621,-41.279,-179.669,5.407,148.843
C06149=1220.315,-10.872,-41.265,-179.672,5.406,148.844
C06150=1220.321,-11.121,-41.251,-179.674,5.406,148.845
C06151=1220.326,-11.370,-41.237,-179.676,5.405,148.845
C06152=1220.330,-11.620,-41.223,-179.679,5.405,148.846
C06153=1220.336,-11.869,-41.210,-179.681,5.405,148.847
C06154=1220.341,-12.119,-41.196,-179.684,5.405,148.847
C06155=1220.346,-12.368,-41.182,-179.686,5.404,148.848
C06156=1220.351,-12.618,-41.169,-179.689,5.404,148.849
C06157=1220.356,-12.868,-41.155,-179.691,5.404,148.849
C06158=1220.361,-13.117,-41.141,-179.694,5.404,148.850
C06159=1220.366,-13.367,-41.126,-179.696,5.403,148.851
C06160=1220.371,-13.617,-41.114,-179.699,5.403,148.852
C06161=1220.377,-13.866,-41.100,-179.701,5.403,148.852
C06162=1220.381,-14.115,-41.085,-179.704,5.402,148.853
C06163=1220.386,-14.365,-41.072,-179.706,5.402,148.854
C06164=1220.392,-14.614,-41.058,-179.709,5.402,148.854
C06165=1220.397,-14.865,-41.045,-179.711,5.402,148.855
C06166=1220.402,-15.114,-41.031,-179.714,5.401,148.856
C06167=1220.407,-15.363,-41.017,-179.716,5.401,148.856
C06168=1220.412,-15.613,-41.004,-179.719,5.401,148.857
C06169=1220.417,-15.862,-40.990,-179.721,5.400,148.858
C06170=1220.422,-16.112,-40.977,-179.724,5.400,148.858
C06171=1220.427,-16.361,-40.963,-179.726,5.400,148.859
C06172=1220.432,-16.611,-40.949,-179.729,5.400,148.860
C06173=1220.437,-16.861,-40.936,-179.731,5.399,148.861
C06174=1220.442,-17.110,-40.922,-179.734,5.399,148.861
C06175=1220.448,-17.361,-40.908,-179.736,5.399,148.862
C06176=1220.453,-17.609,-40.895,-179.739,5.399,148.863
C06177=1220.458,-17.860,-40.881,-179.741,5.398,148.863
C06178=1220.463,-18.108,-40.868,-179.743,5.398,148.864
C06179=1220.468,-18.359,-40.854,-179.746,5.398,148.865
C06180=1220.473,-18.608,-40.840,-179.749,5.397,148.865
C06181=1220.478,-18.858,-40.828,-179.751,5.398,148.866
C06182=1220.483,-19.107,-40.813,-179.753,5.397,148.867
C06183=1220.488,-19.357,-40.801,-179.756,5.397,148.867
C06184=1220.493,-19.606,-40.786,-179.758,5.396,148.868
C06185=1220.499,-19.856,-40.773,-179.760,5.396,148.869
C06186=1220.503,-20.105,-40.760,-179.763,5.396,148.869
C06187=1220.509,-20.355,-40.746,-179.766,5.395,148.870
C06188=1220.513,-20.604,-40.733,-179.768,5.395,148.871
C06189=1220.519,-20.854,-40.719,-179.770,5.395,148.871
C06190=1220.523,-21.103,-40.706,-179.773,5.394,148.872
C06191=1220.529,-21.353,-40.693,-179.775,5.395,148.873
C06192=1220.534,-21.603,-40.678,-179.778,5.394,148.873
C06193=1220.539,-21.853,-40.665,-179.780,5.394,148.874
C06194=1220.544,-22.102,-40.652,-179.783,5.393,148.875
C06195=1220.549,-22.372,-40.638,-179.785,5.394,148.876
C06196=1220.555,-22.640,-40.623,-179.788,5.393,148.877
C06197=1220.561,-22.910,-40.609,-179.791,5.393,148.877
C06198=1220.566,-23.179,-40.594,-179.794,5.392,148.878
C06199=1220.571,-23.429,-40.581,-179.796,5.393,148.879
C06200=1220.576,-23.678,-40.568,-179.798,5.392,148.879
C06201=1220.582,-23.928,-40.554,-179.801,5.392,148.880
C06202=1220.586,-24.178,-40.541,-179.804,5.391,148.881
C06203=1220.592,-24.427,-40.528,-179.806,5.392,148.881
C06204=1220.596,-24.677,-40.515,-179.809,5.391,148.882
C06205=1220.602,-24.927,-40.501,-179.811,5.391,148.883
C06206=1220.606,-25.176,-40.488,-179.813,5.391,148.883
C06207=1220.612,-25.426,-40.474,-179.816,5.390,148.884
C06208=1220.617,-25.676,-40.462,-179.819,5.390,148.885
C06209=1220.622,-25.925,-40.448,-179.821,5.390,148.886
C06210=1220.627,-26.175,-40.435,-179.823,5.390,148.886
C06211=1220.633,-26.424,-40.421,-179.826,5.389,148.887
C06212=1220.637,-26.674,-40.408,-179.828,5.390,148.888
C06213=1220.642,-26.923,-40.395,-179.831,5.389,148.888
C06214=1220.648,-27.173,-40.382,-179.833,5.389,148.889
C06215=1220.652,-27.423,-40.369,-179.835,5.389,148.890
C06216=1220.658,-27.672,-40.356,-179.838,5.388,148.890
C06217=1220.662,-27.922,-40.342,-179.841,5.388,148.891
C06218=1220.667,-28.171,-40.330,-179.843,5.388,148.892
C06219=1220.673,-28.422,-40.316,-179.846,5.388,148.893
C06220=1220.678,-28.671,-40.303,-179.848,5.387,148.893
C06221=1220.683,-28.920,-40.289,-179.850,5.387,148.894
C06222=1220.688,-29.170,-40.276,-179.852,5.387,148.894
C06223=1220.693,-29.419,-40.264,-179.855,5.386,148.895
C06224=1220.698,-29.669,-40.250,-179.857,5.387,148.896
C06225=1220.703,-29.919,-40.238,-179.860,5.386,148.896
C06226=1220.709,-30.168,-40.225,-179.862,5.386,148.897
C06227=1220.714,-30.418,-40.211,-179.865,5.386,148.898
C06228=1220.719,-30.667,-40.198,-179.867,5.385,148.899
C06229=1220.724,-30.917,-40.185,-179.870,5.385,148.899
C06230=1220.729,-31.167,-40.172,-179.872,5.385,148.900
C06231=1220.734,-31.416,-40.159,-179.875,5.385,148.901
C06232=1220.739,-31.666,-40.146,-179.877,5.384,148.901
C06233=1220.745,-31.916,-40.133,-179.879,5.385,148.902
C06234=1220.749,-32.166,-40.120,-179.882,5.384,148.903
C06235=1220.754,-32.414,-40.107,-179.885,5.384,148.903
C06236=1220.760,-32.664,-40.094,-179.887,5.384,148.904
C06237=1220.764,-32.914,-40.081,-179.889,5.383,148.905
C06238=1220.769,-33.163,-40.068,-179.892,5.383,148.906
C06239=1220.775,-33.413,-40.055,-179.894,5.383,148.906
C06240=1220.780,-33.663,-40.042,-179.897,5.383,148.907
C06241=1220.785,-33.912,-40.029,-179.900,5.382,148.908
C06242=1220.791,-34.162,-40.016,-179.902,5.383,148.908
C06243=1220.795,-34.412,-40.003,-179.904,5.382,148.909
C06244=1220.800,-34.661,-39.991,-179.907,5.382,148.910
C06245=1220.806,-34.911,-39.978,-179.909,5.382,148.910
C06246=1220.811,-35.161,-39.965,-179.912,5.381,148.911
C06247=1220.816,-35.410,-39.952,-179.914,5.382,148.912
C06248=1220.821,-35.660,-39.939,-179.916,5.381,148.913
C06249=1220.826,-35.910,-39.926,-179.919,5.381,148.913
C06250=1220.831,-36.159,-39.913,-179.921,5.381,148.914
C06251=1220.837,-36.409,-39.901,-179.924,5.381,148.915
C06252=1220.841,-36.659,-39.888,-179.926,5.380,148.915
C06253=1220.846,-36.908,-39.875,-179.929,5.381,148.916
C06254=1220.852,-37.158,-39.862,-179.931,5.380,148.917
C06255=1220.857,-37.407,-39.849,-179.934,5.380,148.917
C06256=1220.862,-37.657,-39.836,-179.936,5.380,148.918
C06257=1220.867,-37.906,-39.824,-179.939,5.379,148.919
C06258=1220.872,-38.156,-39.811,-179.941,5.379,148.920
C06259=1220.877,-38.406,-39.798,-179.943,5.379,148.920
C06260=1220.882,-38.655,-39.785,-179.946,5.379,148.921
C06261=1220.887,-38.905,-39.772,-179.948,5.379,148.922
C06262=1220.893,-39.154,-39.760,-179.951,5.379,148.922
C06263=1220.897,-39.404,-39.747,-179.953,5.378,148.923
C06264=1220.903,-39.654,-39.735,-179.956,5.378,148.924
C06265=1220.908,-39.903,-39.722,-179.958,5.378,148.924
C06266=1220.914,-40.153,-39.709,-179.960,5.377,148.925
C06267=1220.918,-40.403,-39.696,-179.962,5.377,148.926
C06268=1220.923,-40.652,-39.683,-179.965,5.377,148.926
C06269=1220.928,-40.901,-39.671,-179.967,5.377,148.927
C06270=1220.934,-41.151,-39.659,-179.970,5.377,148.928
C06271=1220.938,-41.401,-39.646,-179.973,5.376,148.928
C06272=1220.943,-41.651,-39.633,-179.975,5.377,148.929
C06273=1220.949,-41.900,-39.620,-179.977,5.376,148.930
C06274=1220.954,-42.150,-39.608,-179.980,5.376,148.931
C06275=1220.959,-42.400,-39.595,-179.982,5.376,148.931
C06276=1220.964,-42.650,-39.583,-179.985,5.376,148.932
C06277=1220.969,-42.899,-39.570,-179.987,5.375,148.933
C06278=1220.975,-43.148,-39.558,-179.989,5.375,148.933
C06279=1220.979,-43.398,-39.545,-179.992,5.375,148.934
C06280=1220.985,-43.648,-39.533,-179.994,5.375,148.935
C06281=1220.990,-43.897,-39.520,-179.997,5.375,148.935
C06282=1220.995,-44.147,-39.508,-180.000,5.374,148.936
C06283=1221.000,-44.396,-39.495,179.998,5.375,148.937
C06284=1221.005,-44.647,-39.483,179.996,5.374,148.938
C06285=1221.011,-44.896,-39.469,179.994,5.374,148.938
C06286=1221.016,-45.146,-39.457,179.991,5.374,148.939
C06287=1221.021,-45.395,-39.444,179.988,5.373,148.940
C06288=1221.026,-45.645,-39.432,179.986,5.374,148.940
C06289=1221.031,-45.894,-39.420,179.984,5.373,148.941
C06290=1221.036,-46.144,-39.407,179.981,5.373,148.942
C06291=1221.041,-46.394,-39.395,179.979,5.373,148.942
C06292=1221.046,-46.644,-39.382,179.976,5.373,148.943
C06293=1221.052,-46.893,-39.370,179.974,5.373,148.944
C06294=1221.057,-47.143,-39.358,179.971,5.373,148.945
C06295=1221.062,-47.392,-39.345,179.969,5.372,148.945
C06296=1221.067,-47.642,-39.332,179.967,5.372,148.946
C06297=1221.072,-47.892,-39.320,179.964,5.372,148.947
C06298=1221.077,-48.141,-39.308,179.962,5.372,148.947
C06299=1221.082,-48.411,-39.294,179.959,5.372,148.948
C06300=1221.088,-48.681,-39.282,179.957,5.371,148.949
C06301=1221.094,-48.951,-39.267,179.954,5.371,148.949
C06302=1221.100,-49.220,-39.255,179.951,5.372,148.950
C06303=1221.104,-49.470,-39.242,179.949,5.371,148.951
C06304=1221.110,-49.720,-39.230,179.946,5.370,148.952
C06305=1221.115,-49.970,-39.217,179.944,5.371,148.952
C06306=1221.120,-50.220,-39.205,179.942,5.370,148.953
C06307=1221.125,-50.469,-39.193,179.940,5.370,148.954
C06308=1221.130,-50.718,-39.181,179.937,5.370,148.954
C06309=1221.135,-50.968,-39.169,179.934,5.369,148.955
C06310=1221.140,-51.217,-39.156,179.932,5.370,148.956
C06311=1221.145,-51.468,-39.144,179.930,5.369,148.957
C06312=1221.150,-51.717,-39.131,179.927,5.370,148.957
C06313=1221.156,-51.967,-39.119,179.925,5.369,148.958
C06314=1221.161,-52.216,-39.107,179.922,5.369,148.959
C06315=1221.166,-52.466,-39.095,179.920,5.369,148.959
C06316=1221.171,-52.716,-39.082,179.917,5.369,148.960
C06317=1221.177,-52.966,-39.071,179.915,5.369,148.961
C06318=1221.181,-53.215,-39.059,179.913,5.368,148.961
C06319=1221.187,-53.465,-39.047,179.910,5.368,148.962
C06320=1221.192,-53.714,-39.034,179.908,5.368,148.963
C06321=1221.197,-53.964,-39.022,179.905,5.368,148.964
C06322=1221.202,-54.213,-39.010,179.903,5.368,148.964
C06323=1221.207,-54.464,-38.997,179.900,5.368,148.965
C06324=1221.212,-54.713,-38.985,179.898,5.367,148.966
C06325=1221.217,-54.963,-38.973,179.896,5.368,148.966
C06326=1221.222,-55.212,-38.961,179.893,5.367,148.967
C06327=1221.228,-55.462,-38.949,179.891,5.367,148.968
C06328=1221.233,-55.712,-38.937,179.888,5.367,148.968
C06329=1221.238,-55.961,-38.924,179.886,5.367,148.969
C06330=1221.243,-56.211,-38.913,179.884,5.367,148.970
C06331=1221.248,-56.460,-38.901,179.881,5.366,148.971
C06332=1221.253,-56.710,-38.889,179.879,5.367,148.971
C06333=1221.259,-56.960,-38.877,179.876,5.366,148.972
C06334=1221.264,-57.209,-38.864,179.874,5.367,148.973
C06335=1221.269,-57.459,-38.853,179.871,5.366,148.973
C06336=1221.274,-57.709,-38.841,179.869,5.366,148.974
C06337=1221.279,-57.958,-38.828,179.867,5.366,148.975
C06338=1221.285,-58.208,-38.816,179.864,5.365,148.975
C06339=1221.289,-58.457,-38.804,179.862,5.366,148.976
C06340=1221.294,-58.707,-38.793,179.860,5.365,148.977
C06341=1221.300,-58.957,-38.781,179.858,5.365,148.977
C06342=1221.305,-59.206,-38.768,179.855,5.365,148.978
C06343=1221.310,-59.456,-38.757,179.852,5.364,148.979
C06344=1221.315,-59.706,-38.745,179.850,5.365,148.980
C06345=1221.320,-59.956,-38.733,179.848,5.364,148.980
C06346=1221.326,-60.205,-38.720,179.845,5.365,148.981
C06347=1221.330,-60.455,-38.709,179.843,5.364,148.982
C06348=1221.336,-60.705,-38.697,179.840,5.364,148.982
C06349=1221.341,-60.954,-38.685,179.838,5.364,148.983
C06350=1221.346,-61.204,-38.673,179.835,5.364,148.984
C06351=1221.351,-61.454,-38.662,179.833,5.364,148.984
C06352=1221.356,-61.704,-38.650,179.831,5.363,148.985
C06353=1221.362,-61.953,-38.637,179.829,5.364,148.986
C06354=1221.366,-62.203,-38.626,179.826,5.363,148.987
C06355=1221.372,-62.452,-38.614,179.823,5.363,148.987
C06356=1221.377,-62.702,-38.602,179.821,5.363,148.988
C06357=1221.382,-62.952,-38.591,179.818,5.363,148.989
C06358=1221.387,-63.201,-38.578,179.816,5.363,148.989
C06359=1221.392,-63.451,-38.566,179.814,5.363,148.990
C06360=1221.397,-63.701,-38.555,179.812,5.363,148.991
C06361=1221.403,-63.950,-38.543,179.809,5.363,148.992
C06362=1221.408,-64.200,-38.531,179.807,5.363,148.992
C06363=1221.413,-64.449,-38.519,179.805,5.362,148.993
C06364=1221.418,-64.699,-38.508,179.802,5.362,148.993
C06365=1221.424,-64.949,-38.496,179.800,5.362,148.994
C06366=1221.428,-65.199,-38.484,179.797,5.361,148.995
C06367=1221.434,-65.449,-38.473,179.795,5.362,148.996
C06368=1221.439,-65.698,-38.461,179.792,5.361,148.996
C06369=1221.444,-65.948,-38.449,179.790,5.362,148.997
C06370=1221.449,-66.197,-38.437,179.788,5.361,148.998
C06371=1221.454,-66.447,-38.425,179.785,5.361,148.998
C06372=1221.460,-66.696,-38.414,179.783,5.361,148.999
C06373=1221.465,-66.946,-38.402,179.780,5.361,149.000
C06374=1221.470,-67.196,-38.391,179.778,5.361,149.000
C06375=1221.475,-67.446,-38.379,179.776,5.361,149.001
C06376=1221.480,-67.695,-38.368,179.773,5.361,149.002
C06377=1221.485,-67.945,-38.356,179.771,5.360,149.003
C06378=1221.490,-68.195,-38.344,179.769,5.361,149.003
C06379=1221.496,-68.445,-38.333,179.766,5.360,149.004
C06380=1221.502,-68.694,-38.321,179.763,5.360,149.005
C06381=1221.506,-68.944,-38.310,179.761,5.360,149.005
C06382=1221.512,-69.194,-38.298,179.759,5.360,149.006
C06383=1221.516,-69.443,-38.287,179.757,5.360,149.007
C06384=1221.522,-69.693,-38.275,179.754,5.360,149.008
C06385=1221.527,-69.943,-38.263,179.752,5.360,149.008
C06386=1221.532,-70.193,-38.251,179.750,5.359,149.009
C06387=1221.537,-70.442,-38.241,179.747,5.360,149.009
C06388=1221.543,-70.692,-38.229,179.745,5.359,149.010
C06389=1221.547,-70.941,-38.217,179.743,5.359,149.011
C06390=1221.553,-71.191,-38.206,179.740,5.359,149.012
C06391=1221.558,-71.441,-38.194,179.737,5.358,149.012
C06392=1221.563,-71.691,-38.182,179.735,5.359,149.013
C06393=1221.568,-71.940,-38.171,179.733,5.358,149.014
C06394=1221.574,-72.190,-38.160,179.731,5.359,149.014
C06395=1221.578,-72.439,-38.148,179.728,5.358,149.015
C06396=1221.584,-72.689,-38.136,179.726,5.359,149.016
C06397=1221.588,-72.939,-38.125,179.723,5.358,149.017
C06398=1221.595,-73.188,-38.114,179.721,5.359,149.017
C06399=1221.599,-73.438,-38.102,179.718,5.358,149.018
C06400=1221.605,-73.688,-38.090,179.716,5.358,149.019
C06401=1221.609,-73.937,-38.079,179.714,5.358,149.019
C06402=1221.615,-74.187,-38.067,179.711,5.358,149.020
C06403=1221.621,-74.457,-38.055,179.709,5.358,149.021
C06404=1221.627,-74.728,-38.043,179.706,5.357,149.021
C06405=1221.631,-74.999,-38.031,179.703,5.357,149.022
C06406=1221.637,-75.269,-38.019,179.701,5.357,149.023
C06407=1221.643,-75.519,-38.007,179.699,5.357,149.024
C06408=1221.647,-75.768,-37.996,179.697,5.357,149.024
C06409=1221.654,-76.018,-37.984,179.694,5.357,149.025
C06410=1221.658,-76.267,-37.973,179.692,5.357,149.026
C06411=1221.663,-76.517,-37.962,179.689,5.357,149.026
C06412=1221.669,-76.767,-37.950,179.687,5.357,149.027
C06413=1221.674,-77.016,-37.939,179.684,5.357,149.028
C06414=1221.679,-77.266,-37.928,179.682,5.356,149.029
C06415=1221.684,-77.516,-37.916,179.680,5.356,149.029
C06416=1221.689,-77.766,-37.906,179.677,5.356,149.030
C06417=1221.695,-78.015,-37.894,179.675,5.356,149.031
C06418=1221.700,-78.265,-37.883,179.672,5.356,149.031
C06419=1221.704,-78.515,-37.872,179.671,5.356,149.032
C06420=1221.710,-78.765,-37.860,179.668,5.355,149.033
C06421=1221.716,-79.014,-37.849,179.666,5.356,149.033
C06422=1221.721,-79.264,-37.838,179.663,5.355,149.034
C06423=1221.726,-79.514,-37.826,179.661,5.356,149.035
C06424=1221.731,-79.763,-37.816,179.658,5.355,149.035
C06425=1221.737,-80.013,-37.804,179.656,5.356,149.036
C06426=1221.741,-80.263,-37.793,179.654,5.355,149.037
C06427=1221.746,-80.512,-37.782,179.652,5.356,149.038
C06428=1221.752,-80.762,-37.771,179.649,5.355,149.038
C06429=1221.757,-81.012,-37.760,179.647,5.355,149.039
C06430=1221.762,-81.261,-37.748,179.644,5.355,149.040
C06431=1221.767,-81.511,-37.738,179.641,5.355,149.040
C06432=1221.773,-81.761,-37.726,179.639,5.355,149.041
C06433=1221.777,-82.011,-37.715,179.637,5.354,149.042
C06434=1221.783,-82.260,-37.705,179.635,5.354,149.042
C06435=1221.789,-82.510,-37.693,179.632,5.354,149.043
C06436=1221.793,-82.760,-37.681,179.630,5.354,149.044
C06437=1221.798,-83.010,-37.671,179.628,5.354,149.044
C06438=1221.803,-83.259,-37.660,179.626,5.354,149.045
C06439=1221.809,-83.509,-37.648,179.623,5.354,149.046
C06440=1221.814,-83.759,-37.638,179.621,5.354,149.047
C06441=1221.819,-84.008,-37.627,179.618,5.354,149.047
C06442=1221.824,-84.258,-37.615,179.616,5.354,149.048
C06443=1221.830,-84.508,-37.604,179.613,5.354,149.049
C06444=1221.835,-84.757,-37.593,179.611,5.354,149.049
C06445=1221.840,-85.007,-37.583,179.609,5.354,149.050
C06446=1221.845,-85.256,-37.572,179.607,5.354,149.051
C06447=1221.850,-85.506,-37.560,179.604,5.353,149.051
C06448=1221.856,-85.756,-37.549,179.602,5.353,149.052
C06449=1221.861,-86.005,-37.538,179.600,5.353,149.053
C06450=1221.866,-86.256,-37.528,179.598,5.353,149.053
C06451=1221.871,-86.505,-37.516,179.595,5.353,149.054
C06452=1221.876,-86.755,-37.506,179.593,5.353,149.055
C06453=1221.882,-87.005,-37.494,179.590,5.353,149.056
C06454=1221.887,-87.255,-37.484,179.588,5.353,149.056
C06455=1221.892,-87.504,-37.473,179.585,5.353,149.057
C06456=1221.897,-87.754,-37.462,179.583,5.353,149.058
C06457=1221.902,-88.003,-37.451,179.581,5.353,149.058
C06458=1221.908,-88.254,-37.440,179.578,5.353,149.059
C06459=1221.913,-88.503,-37.429,179.576,5.352,149.060
C06460=1221.918,-88.753,-37.419,179.574,5.353,149.060
C06461=1221.923,-89.002,-37.407,179.572,5.352,149.061
C06462=1221.929,-89.252,-37.397,179.569,5.352,149.062
C06463=1221.933,-89.502,-37.386,179.567,5.352,149.062
C06464=1221.938,-89.752,-37.375,179.564,5.352,149.063
C06465=1221.944,-90.001,-37.364,179.562,5.352,149.064
C06466=1221.949,-90.251,-37.353,179.559,5.351,149.065
C06467=1221.955,-90.500,-37.342,179.557,5.352,149.065
C06468=1221.960,-90.750,-37.332,179.555,5.351,149.066
C06469=1221.965,-90.999,-37.321,179.552,5.352,149.067
C06470=1221.970,-91.250,-37.310,179.550,5.351,149.067
C06471=1221.975,-91.500,-37.300,179.548,5.351,149.068
C06472=1221.980,-91.749,-37.289,179.546,5.351,149.069
C06473=1221.985,-91.999,-37.278,179.543,5.351,149.069
C06474=1221.991,-92.248,-37.267,179.541,5.351,149.070
C06475=1221.996,-92.499,-37.256,179.539,5.351,149.071
C06476=1222.002,-92.748,-37.246,179.536,5.351,149.071
C06477=1222.006,-92.998,-37.235,179.534,5.351,149.072
C06478=1222.012,-93.247,-37.224,179.531,5.351,149.073
C06479=1222.017,-93.497,-37.214,179.529,5.351,149.074
C06480=1222.022,-93.746,-37.203,179.527,5.350,149.074
C06481=1222.027,-93.997,-37.192,179.525,5.351,149.075
C06482=1222.033,-94.246,-37.182,179.522,5.350,149.075
C06483=1222.038,-94.496,-37.171,179.520,5.350,149.076
C06484=1222.043,-94.746,-37.160,179.517,5.350,149.077
C06485=1222.048,-94.996,-37.150,179.515,5.350,149.078
C06486=1222.053,-95.245,-37.139,179.513,5.350,149.078
C06487=1222.059,-95.495,-37.129,179.511,5.350,149.079
C06488=1222.064,-95.745,-37.118,179.508,5.350,149.080
C06489=1222.069,-95.994,-37.107,179.506,5.350,149.080
C06490=1222.074,-96.244,-37.096,179.504,5.349,149.081
C06491=1222.079,-96.494,-37.086,179.502,5.350,149.082
C06492=1222.084,-96.744,-37.076,179.499,5.349,149.082
C06493=1222.090,-96.993,-37.065,179.497,5.350,149.083
C06494=1222.095,-97.242,-37.055,179.495,5.350,149.084
C06495=1222.100,-97.493,-37.044,179.492,5.350,149.085
C06496=1222.106,-97.742,-37.034,179.490,5.350,149.085
C06497=1222.111,-97.992,-37.022,179.487,5.350,149.086
C06498=1222.116,-98.241,-37.012,179.486,5.350,149.086
C06499=1222.121,-98.492,-37.002,179.483,5.349,149.087
C06500=1222.127,-98.741,-36.991,179.481,5.350,149.088
C06501=1222.131,-98.991,-36.980,179.478,5.349,149.089
C06502=1222.137,-99.240,-36.970,179.476,5.349,149.089
C06503=1222.142,-99.491,-36.959,179.473,5.349,149.090
C06504=1222.148,-99.740,-36.949,179.471,5.349,149.091
C06505=1222.153,-99.990,-36.939,179.469,5.349,149.091
C06506=1222.158,-100.239,-36.928,179.467,5.349,149.092
C06507=1222.163,-100.511,-36.917,179.464,5.349,149.093
C06508=1222.170,-100.781,-36.906,179.461,5.348,149.094
C06509=1222.175,-101.053,-36.895,179.459,5.349,149.094
C06510=1222.180,-101.324,-36.882,179.456,5.348,149.095
C06511=1222.186,-101.573,-36.872,179.454,5.349,149.096
C06512=1222.191,-101.824,-36.862,179.452,5.348,149.096
C06513=1222.197,-102.073,-36.851,179.450,5.349,149.097
C06514=1222.201,-102.323,-36.841,179.447,5.348,149.098
C06515=1222.207,-102.573,-36.831,179.445,5.348,149.098
C06516=1222.212,-102.822,-36.821,179.443,5.348,149.099
C06517=1222.217,-103.072,-36.810,179.441,5.348,149.100
C06518=1222.223,-103.322,-36.800,179.438,5.348,149.100
C06519=1222.227,-103.572,-36.789,179.436,5.348,149.101
C06520=1222.233,-103.821,-36.779,179.433,5.348,149.102
C06521=1222.239,-104.071,-36.769,179.431,5.348,149.103
C06522=1222.243,-104.321,-36.759,179.428,5.348,149.103
C06523=1222.248,-104.570,-36.748,179.427,5.348,149.104
C06524=1222.253,-104.820,-36.738,179.424,5.347,149.105
C06525=1222.259,-105.070,-36.728,179.422,5.348,149.105
C06526=1222.265,-105.319,-36.717,179.419,5.347,149.106
C06527=1222.270,-105.570,-36.707,179.417,5.348,149.107
C06528=1222.274,-105.819,-36.697,179.415,5.348,149.107
C06529=1222.280,-106.068,-36.687,179.412,5.347,149.108
C06530=1222.285,-106.319,-36.676,179.411,5.347,149.109
C06531=1222.291,-106.568,-36.666,179.408,5.347,149.109
C06532=1222.296,-106.818,-36.656,179.406,5.347,149.110
C06533=1222.301,-107.068,-36.646,179.403,5.347,149.111
C06534=1222.306,-107.317,-36.636,179.401,5.347,149.111
C06535=1222.311,-107.568,-36.625,179.399,5.347,149.112
C06536=1222.317,-107.817,-36.615,179.397,5.347,149.113
C06537=1222.322,-108.067,-36.605,179.394,5.346,149.113
C06538=1222.327,-108.317,-36.595,179.392,5.347,149.114
C06539=1222.332,-108.566,-36.585,179.390,5.346,149.115
C06540=1222.338,-108.816,-36.574,179.387,5.347,149.115
C06541=1222.343,-109.066,-36.564,179.385,5.346,149.116
C06542=1222.348,-109.315,-36.554,179.383,5.347,149.117
C06543=1222.353,-109.565,-36.544,179.380,5.346,149.118
C06544=1222.358,-109.815,-36.533,179.378,5.346,149.118
C06545=1222.364,-110.065,-36.524,179.376,5.346,149.119
C06546=1222.369,-110.314,-36.514,179.374,5.346,149.120
C06547=1222.374,-110.565,-36.504,179.372,5.347,149.120
C06548=1222.380,-110.814,-36.494,179.369,5.346,149.121
C06549=1222.385,-111.064,-36.483,179.367,5.347,149.122
C06550=1222.390,-111.313,-36.474,179.364,5.346,149.122
C06551=1222.395,-111.563,-36.463,179.363,5.346,149.123
C06552=1222.401,-111.813,-36.453,179.360,5.346,149.124
C06553=1222.406,-112.062,-36.444,179.358,5.346,149.124
C06554=1222.411,-112.313,-36.433,179.355,5.346,149.125
C06555=1222.416,-112.562,-36.423,179.353,5.346,149.126
C06556=1222.421,-112.811,-36.414,179.350,5.346,149.126
C06557=1222.427,-113.061,-36.403,179.349,5.346,149.127
C06558=1222.432,-113.311,-36.393,179.346,5.345,149.128
C06559=1222.437,-113.561,-36.384,179.344,5.346,149.128
C06560=1222.443,-113.811,-36.374,179.341,5.345,149.129
C06561=1222.448,-114.061,-36.363,179.339,5.346,149.130
C06562=1222.453,-114.310,-36.354,179.337,5.346,149.131
C06563=1222.458,-114.560,-36.343,179.335,5.345,149.131
C06564=1222.464,-114.810,-36.334,179.333,5.346,149.132
C06565=1222.468,-115.060,-36.324,179.330,5.345,149.132
C06566=1222.474,-115.309,-36.314,179.328,5.345,149.133
C06567=1222.479,-115.559,-36.303,179.325,5.345,149.134
C06568=1222.484,-115.808,-36.294,179.323,5.345,149.135
C06569=1222.490,-116.059,-36.284,179.321,5.345,149.135
C06570=1222.495,-116.309,-36.274,179.319,5.345,149.136
C06571=1222.500,-116.558,-36.264,179.316,5.345,149.137
C06572=1222.506,-116.808,-36.255,179.314,5.345,149.137
C06573=1222.511,-117.057,-36.245,179.312,5.345,149.138
C06574=1222.516,-117.307,-36.234,179.309,5.345,149.139
C06575=1222.521,-117.557,-36.224,179.308,5.345,149.139
C06576=1222.527,-117.807,-36.215,179.305,5.344,149.140
C06577=1222.532,-118.056,-36.205,179.303,5.345,149.141
C06578=1222.536,-118.306,-36.195,179.300,5.344,149.141
C06579=1222.542,-118.556,-36.186,179.298,5.345,149.142
C06580=1222.548,-118.806,-36.175,179.296,5.344,149.142
C06581=1222.553,-119.055,-36.166,179.294,5.344,149.143
C06582=1222.559,-119.305,-36.156,179.291,5.344,149.144
C06583=1222.563,-119.555,-36.146,179.289,5.344,149.145
C06584=1222.569,-119.805,-36.136,179.287,5.344,149.145
C06585=1222.574,-120.055,-36.127,179.285,5.344,149.146
C06586=1222.579,-120.304,-36.117,179.283,5.344,149.147
C06587=1222.584,-120.553,-36.107,179.280,5.344,149.147
C06588=1222.590,-120.804,-36.098,179.278,5.344,149.148
C06589=1222.594,-121.054,-36.088,179.275,5.344,149.149
C06590=1222.600,-121.303,-36.078,179.273,5.344,149.149
C06591=1222.605,-121.553,-36.069,179.271,5.343,149.150
C06592=1222.611,-121.802,-36.059,179.269,5.344,149.151
C06593=1222.616,-122.052,-36.050,179.266,5.343,149.151
C06594=1222.622,-122.302,-36.040,179.264,5.344,149.152
C06595=1222.626,-122.552,-36.030,179.262,5.343,149.153
C06596=1222.632,-122.802,-36.020,179.260,5.343,149.153
C06597=1222.637,-123.051,-36.010,179.258,5.344,149.154
C06598=1222.642,-123.301,-36.001,179.255,5.343,149.155
C06599=1222.647,-123.551,-35.991,179.253,5.344,149.155
C06600=1222.653,-123.801,-35.982,179.250,5.343,149.156
C06601=1222.658,-124.050,-35.972,179.249,5.343,149.157
C06602=1222.663,-124.301,-35.962,179.246,5.343,149.157
C06603=1222.668,-124.550,-35.953,179.244,5.343,149.158
C06604=1222.674,-124.800,-35.943,179.241,5.343,149.159
C06605=1222.679,-125.050,-35.934,179.239,5.343,149.159
C06606=1222.685,-125.300,-35.924,179.237,5.342,149.160
C06607=1222.690,-125.549,-35.915,179.235,5.343,149.161
C06608=1222.696,-125.799,-35.905,179.233,5.343,149.161
C06609=1222.701,-126.048,-35.895,179.230,5.343,149.162
C06610=1222.705,-126.299,-35.886,179.229,5.343,149.163
C06611=1222.285,-126.309,-35.922,179.224,5.346,149.165
C06612=1222.279,-126.059,-35.932,179.226,5.346,149.164
C06613=1222.274,-125.810,-35.941,179.229,5.346,149.163
C06614=1222.268,-125.560,-35.951,179.231,5.346,149.163
C06615=1222.263,-125.310,-35.961,179.233,5.346,149.162
C06616=1222.257,-125.060,-35.970,179.235,5.346,149.161
C06617=1222.252,-124.811,-35.980,179.237,5.346,149.161
C06618=1222.246,-124.561,-35.989,179.240,5.346,149.160
C06619=1222.242,-124.312,-35.999,179.242,5.346,149.159
C06620=1222.237,-124.061,-36.008,179.244,5.347,149.159
C06621=1222.231,-123.812,-36.018,179.246,5.346,149.158
C06622=1222.226,-123.562,-36.027,179.249,5.347,149.157
C06623=1222.221,-123.312,-36.037,179.251,5.347,149.157
C06624=1222.216,-123.062,-36.046,179.253,5.347,149.156
C06625=1222.210,-122.813,-36.056,179.256,5.347,149.155
C06626=1222.205,-122.564,-36.066,179.258,5.347,149.155
C06627=1222.200,-122.313,-36.076,179.260,5.347,149.154
C06628=1222.195,-122.063,-36.086,179.262,5.347,149.153
C06629=1222.189,-121.813,-36.095,179.265,5.347,149.153
C06630=1222.184,-121.564,-36.105,179.267,5.347,149.152
C06631=1222.178,-121.314,-36.114,179.269,5.347,149.151
C06632=1222.173,-121.065,-36.124,179.271,5.347,149.151
C06633=1222.168,-120.814,-36.134,179.274,5.348,149.150
C06634=1222.163,-120.565,-36.143,179.276,5.347,149.149
C06635=1222.158,-120.315,-36.153,179.278,5.347,149.149
C06636=1222.153,-120.066,-36.163,179.280,5.347,149.148
C06637=1222.147,-119.816,-36.173,179.283,5.347,149.147
C06638=1222.141,-119.566,-36.183,179.285,5.348,149.147
C06639=1222.137,-119.315,-36.192,179.287,5.348,149.146
C06640=1222.131,-119.066,-36.202,179.290,5.348,149.145
C06641=1222.126,-118.817,-36.212,179.292,5.348,149.145
C06642=1222.120,-118.567,-36.221,179.294,5.348,149.144
C06643=1222.115,-118.317,-36.231,179.296,5.348,149.143
C06644=1222.110,-118.067,-36.241,179.299,5.348,149.143
C06645=1222.105,-117.818,-36.252,179.301,5.348,149.142
C06646=1222.100,-117.568,-36.261,179.303,5.348,149.141
C06647=1222.094,-117.318,-36.271,179.305,5.348,149.141
C06648=1222.090,-117.068,-36.281,179.308,5.348,149.140
C06649=1222.084,-116.818,-36.290,179.310,5.348,149.139
C06650=1222.079,-116.569,-36.300,179.312,5.348,149.139
C06651=1222.073,-116.319,-36.310,179.315,5.349,149.138
C06652=1222.068,-116.070,-36.320,179.317,5.348,149.137
C06653=1222.063,-115.819,-36.330,179.319,5.349,149.136
C06654=1222.058,-115.570,-36.340,179.321,5.348,149.136
C06655=1222.052,-115.320,-36.350,179.324,5.349,149.135
C06656=1222.047,-115.071,-36.360,179.326,5.349,149.135
C06657=1222.042,-114.820,-36.369,179.328,5.349,149.134
C06658=1222.036,-114.570,-36.380,179.330,5.349,149.133
C06659=1222.031,-114.321,-36.389,179.333,5.349,149.132
C06660=1222.026,-114.072,-36.400,179.335,5.349,149.132
C06661=1222.021,-113.821,-36.409,179.337,5.349,149.131
C06662=1222.016,-113.572,-36.419,179.339,5.349,149.130
C06663=1222.010,-113.322,-36.429,179.342,5.349,149.130
C06664=1222.005,-113.072,-36.439,179.344,5.349,149.129
C06665=1222.000,-112.823,-36.449,179.346,5.349,149.128
C06666=1221.995,-112.573,-36.460,179.349,5.349,149.128
C06667=1221.989,-112.323,-36.469,179.351,5.349,149.127
C06668=1221.985,-112.073,-36.479,179.353,5.350,149.126
C06669=1221.979,-111.823,-36.489,179.355,5.349,149.126
C06670=1221.973,-111.574,-36.499,179.358,5.350,149.125
C06671=1221.968,-111.325,-36.509,179.360,5.349,149.124
C06672=1221.963,-111.074,-36.520,179.363,5.350,149.124
C06673=1221.958,-110.825,-36.530,179.364,5.350,149.123
C06674=1221.952,-110.575,-36.539,179.367,5.350,149.122
C06675=1221.948,-110.325,-36.549,179.369,5.350,149.122
C06676=1221.942,-110.075,-36.560,179.371,5.349,149.121
C06677=1221.936,-109.826,-36.570,179.374,5.350,149.120
C06678=1221.931,-109.575,-36.580,179.376,5.349,149.120
C06679=1221.927,-109.326,-36.590,179.379,5.350,149.119
C06680=1221.921,-109.077,-36.600,179.380,5.350,149.118
C06681=1221.916,-108.826,-36.611,179.383,5.350,149.118
C06682=1221.910,-108.577,-36.621,179.385,5.350,149.117
C06683=1221.906,-108.328,-36.631,179.388,5.350,149.116
C06684=1221.901,-108.077,-36.641,179.390,5.350,149.115
C06685=1221.895,-107.828,-36.651,179.393,5.350,149.115
C06686=1221.889,-107.578,-36.662,179.394,5.350,149.114
C06687=1221.885,-107.328,-36.672,179.397,5.351,149.114
C06688=1221.879,-107.078,-36.681,179.399,5.351,149.113
C06689=1221.874,-106.829,-36.691,179.402,5.351,149.112
C06690=1221.869,-106.578,-36.702,179.404,5.351,149.111
C06691=1221.863,-106.329,-36.712,179.406,5.351,149.111
C06692=1221.858,-106.080,-36.722,179.408,5.351,149.110
C06693=1221.853,-105.829,-36.732,179.411,5.351,149.109
C06694=1221.848,-105.580,-36.742,179.413,5.351,149.109
C06695=1221.842,-105.331,-36.753,179.415,5.351,149.108
C06696=1221.837,-105.081,-36.764,179.418,5.351,149.107
C06697=1221.832,-104.831,-36.774,179.420,5.351,149.107
C06698=1221.827,-104.581,-36.784,179.422,5.351,149.106
C06699=1221.822,-104.332,-36.794,179.424,5.351,149.105
C06700=1221.816,-104.082,-36.805,179.427,5.351,149.104
C06701=1221.811,-103.832,-36.815,179.429,5.351,149.104
C06702=1221.806,-103.582,-36.825,179.431,5.352,149.103
C06703=1221.801,-103.332,-36.836,179.433,5.351,149.103
C06704=1221.796,-103.083,-36.845,179.436,5.352,149.102
C06705=1221.790,-102.833,-36.856,179.438,5.351,149.101
C06706=1221.785,-102.583,-36.866,179.441,5.352,149.100
C06707=1221.780,-102.333,-36.876,179.443,5.351,149.100
C06708=1221.775,-102.083,-36.887,179.445,5.352,149.099
C06709=1221.769,-101.834,-36.898,179.447,5.352,149.099
C06710=1221.764,-101.585,-36.908,179.450,5.352,149.098
C06711=1221.759,-101.335,-36.919,179.452,5.352,149.097
C06712=1221.754,-101.063,-36.930,179.455,5.352,149.096
C06713=1221.747,-100.792,-36.941,179.457,5.352,149.096
C06714=1221.742,-100.522,-36.953,179.459,5.352,149.095
C06715=1221.736,-100.250,-36.964,179.463,5.352,149.094
C06716=1221.731,-100.001,-36.974,179.464,5.352,149.094
C06717=1221.726,-99.751,-36.984,179.467,5.353,149.093
C06718=1221.721,-99.501,-36.994,179.469,5.353,149.092
C06719=1221.716,-99.251,-37.006,179.472,5.353,149.091
C06720=1221.710,-99.002,-37.016,179.474,5.353,149.091
C06721=1221.705,-98.752,-37.026,179.476,5.353,149.090
C06722=1221.700,-98.502,-37.037,179.479,5.353,149.089
C06723=1221.694,-98.253,-37.047,179.481,5.353,149.089
C06724=1221.690,-98.003,-37.058,179.483,5.353,149.088
C06725=1221.684,-97.753,-37.068,179.485,5.354,149.087
C06726=1221.679,-97.503,-37.079,179.488,5.353,149.087
C06727=1221.673,-97.254,-37.089,179.490,5.354,149.086
C06728=1221.669,-97.004,-37.101,179.492,5.353,149.085
C06729=1221.663,-96.754,-37.111,179.495,5.354,149.084
C06730=1221.658,-96.504,-37.121,179.497,5.353,149.084
C06731=1221.652,-96.255,-37.132,179.500,5.354,149.083
C06732=1221.648,-96.005,-37.143,179.502,5.353,149.082
C06733=1221.642,-95.755,-37.153,179.503,5.353,149.082
C06734=1221.637,-95.505,-37.164,179.506,5.354,149.081
C06735=1221.632,-95.256,-37.174,179.508,5.353,149.080
C06736=1221.627,-95.006,-37.185,179.511,5.354,149.080
C06737=1221.621,-94.756,-37.195,179.513,5.354,149.079
C06738=1221.616,-94.506,-37.206,179.516,5.354,149.078
C06739=1221.611,-94.257,-37.217,179.518,5.354,149.078
C06740=1221.606,-94.007,-37.227,179.520,5.354,149.077
C06741=1221.600,-93.758,-37.238,179.523,5.354,149.076
C06742=1221.596,-93.508,-37.249,179.525,5.354,149.075
C06743=1221.590,-93.258,-37.259,179.527,5.354,149.075
C06744=1221.584,-93.008,-37.270,179.529,5.355,149.074
C06745=1221.579,-92.759,-37.281,179.532,5.354,149.074
C06746=1221.574,-92.509,-37.292,179.534,5.355,149.073
C06747=1221.569,-92.260,-37.303,179.536,5.354,149.072
C06748=1221.564,-92.009,-37.313,179.539,5.355,149.071
C06749=1221.559,-91.759,-37.324,179.541,5.354,149.071
C06750=1221.554,-91.510,-37.335,179.544,5.355,149.070
C06751=1221.549,-91.260,-37.345,179.546,5.354,149.069
C06752=1221.543,-91.011,-37.356,179.549,5.355,149.069
C06753=1221.538,-90.761,-37.367,179.551,5.356,149.068
C06754=1221.533,-90.511,-37.377,179.553,5.355,149.067
C06755=1221.527,-90.261,-37.389,179.555,5.356,149.067
C06756=1221.522,-90.012,-37.399,179.558,5.355,149.066
C06757=1221.517,-89.762,-37.410,179.560,5.356,149.065
C06758=1221.512,-89.512,-37.421,179.562,5.356,149.065
C06759=1221.507,-89.263,-37.432,179.565,5.356,149.064
C06760=1221.502,-89.013,-37.442,179.567,5.356,149.063
C06761=1221.496,-88.764,-37.453,179.570,5.356,149.062
C06762=1221.491,-88.513,-37.465,179.572,5.356,149.062
C06763=1221.486,-88.264,-37.476,179.574,5.356,149.061
C06764=1221.480,-88.014,-37.486,179.576,5.356,149.061
C06765=1221.476,-87.765,-37.497,179.579,5.357,149.060
C06766=1221.470,-87.515,-37.508,179.581,5.356,149.059
C06767=1221.465,-87.265,-37.519,179.584,5.357,149.058
C06768=1221.460,-87.015,-37.530,179.586,5.356,149.058
C06769=1221.454,-86.766,-37.541,179.588,5.357,149.057
C06770=1221.449,-86.516,-37.552,179.590,5.356,149.056
C06771=1221.445,-86.266,-37.563,179.593,5.357,149.056
C06772=1221.439,-86.016,-37.573,179.595,5.356,149.055
C06773=1221.434,-85.767,-37.584,179.598,5.357,149.054
C06774=1221.428,-85.517,-37.595,179.600,5.357,149.053
C06775=1221.423,-85.267,-37.606,179.602,5.357,149.053
C06776=1221.419,-85.018,-37.618,179.604,5.357,149.052
C06777=1221.413,-84.768,-37.628,179.607,5.357,149.051
C06778=1221.408,-84.518,-37.640,179.609,5.357,149.051
C06779=1221.403,-84.268,-37.650,179.612,5.358,149.050
C06780=1221.397,-84.019,-37.661,179.614,5.357,149.049
C06781=1221.393,-83.769,-37.673,179.616,5.358,149.049
C06782=1221.387,-83.519,-37.684,179.618,5.357,149.048
C06783=1221.382,-83.270,-37.695,179.621,5.358,149.047
C06784=1221.377,-83.020,-37.705,179.623,5.357,149.047
C06785=1221.372,-82.770,-37.717,179.626,5.358,149.046
C06786=1221.366,-82.521,-37.728,179.628,5.357,149.045
C06787=1221.361,-82.271,-37.739,179.630,5.358,149.045
C06788=1221.356,-82.021,-37.750,179.633,5.359,149.044
C06789=1221.351,-81.772,-37.761,179.635,5.358,149.043
C06790=1221.345,-81.522,-37.772,179.638,5.359,149.042
C06791=1221.340,-81.272,-37.783,179.640,5.358,149.042
C06792=1221.335,-81.023,-37.794,179.642,5.359,149.041
C06793=1221.329,-80.772,-37.805,179.644,5.359,149.040
C06794=1221.325,-80.523,-37.817,179.647,5.359,149.040
C06795=1221.320,-80.273,-37.828,179.649,5.359,149.039
C06796=1221.314,-80.024,-37.839,179.652,5.359,149.038
C06797=1221.309,-79.774,-37.850,179.654,5.359,149.038
C06798=1221.304,-79.524,-37.861,179.657,5.359,149.037
C06799=1221.298,-79.275,-37.873,179.659,5.359,149.036
C06800=1221.294,-79.025,-37.884,179.661,5.359,149.035
C06801=1221.289,-78.775,-37.895,179.663,5.359,149.035
C06802=1221.283,-78.525,-37.907,179.666,5.360,149.034
C06803=1221.278,-78.276,-37.918,179.668,5.359,149.034
C06804=1221.273,-78.026,-37.929,179.670,5.360,149.033
C06805=1221.267,-77.776,-37.940,179.673,5.359,149.032
C06806=1221.263,-77.526,-37.951,179.675,5.360,149.031
C06807=1221.257,-77.277,-37.962,179.678,5.360,149.031
C06808=1221.252,-77.027,-37.974,179.680,5.360,149.030
C06809=1221.247,-76.778,-37.985,179.683,5.360,149.029
C06810=1221.242,-76.527,-37.997,179.685,5.360,149.029
C06811=1221.236,-76.278,-38.007,179.687,5.361,149.028
C06812=1221.232,-76.029,-38.019,179.689,5.360,149.027
C06813=1221.226,-75.779,-38.031,179.692,5.361,149.026
C06814=1221.221,-75.529,-38.042,179.694,5.360,149.026
C06815=1221.215,-75.280,-38.053,179.697,5.361,149.025
C06816=1221.210,-75.009,-38.066,179.700,5.361,149.024
C06817=1221.205,-74.738,-38.077,179.702,5.361,149.024
C06818=1221.199,-74.469,-38.090,179.704,5.361,149.023
C06819=1221.193,-74.198,-38.102,179.707,5.362,149.022
C06820=1221.188,-73.948,-38.114,179.709,5.361,149.021
C06821=1221.183,-73.699,-38.125,179.712,5.362,149.021
C06822=1221.177,-73.449,-38.137,179.714,5.362,149.020
C06823=1221.173,-73.199,-38.148,179.717,5.362,149.019
C06824=1221.167,-72.949,-38.160,179.719,5.362,149.019
C06825=1221.162,-72.699,-38.171,179.721,5.362,149.018
C06826=1221.157,-72.450,-38.182,179.723,5.362,149.017
C06827=1221.151,-72.200,-38.193,179.726,5.362,149.016
C06828=1221.147,-71.951,-38.205,179.728,5.362,149.016
C06829=1221.141,-71.701,-38.217,179.731,5.362,149.015
C06830=1221.137,-71.451,-38.228,179.734,5.363,149.014
C06831=1221.131,-71.202,-38.239,179.736,5.362,149.014
C06832=1221.126,-70.952,-38.251,179.738,5.363,149.013
C06833=1221.120,-70.702,-38.263,179.740,5.363,149.012
C06834=1221.115,-70.452,-38.275,179.743,5.363,149.012
C06835=1221.110,-70.203,-38.286,179.745,5.363,149.011
C06836=1221.105,-69.953,-38.298,179.747,5.363,149.010
C06837=1221.100,-69.704,-38.309,179.749,5.363,149.010
C06838=1221.094,-69.454,-38.321,179.752,5.364,149.009
C06839=1221.090,-69.204,-38.332,179.754,5.363,149.008
C06840=1221.084,-68.954,-38.344,179.757,5.364,149.008
C06841=1221.079,-68.705,-38.355,179.759,5.364,149.007
C06842=1221.074,-68.455,-38.367,179.762,5.364,149.006
C06843=1221.069,-68.205,-38.378,179.764,5.364,149.005
C06844=1221.063,-67.956,-38.390,179.766,5.364,149.005
C06845=1221.058,-67.706,-38.402,179.769,5.364,149.004
C06846=1221.053,-67.456,-38.413,179.771,5.364,149.003
C06847=1221.048,-67.206,-38.425,179.774,5.364,149.003
C06848=1221.043,-66.957,-38.437,179.776,5.364,149.002
C06849=1221.038,-66.707,-38.449,179.778,5.365,149.001
C06850=1221.033,-66.458,-38.460,179.781,5.365,149.000
C06851=1221.028,-66.208,-38.472,179.783,5.365,149.000
C06852=1221.022,-65.958,-38.484,179.785,5.366,148.999
C06853=1221.017,-65.709,-38.495,179.788,5.365,148.999
C06854=1221.012,-65.459,-38.507,179.790,5.366,148.998
C06855=1221.006,-65.209,-38.518,179.792,5.365,148.997
C06856=1221.002,-64.960,-38.530,179.795,5.366,148.996
C06857=1220.996,-64.710,-38.542,179.798,5.366,148.996
C06858=1220.992,-64.461,-38.554,179.800,5.366,148.995
C06859=1220.986,-64.211,-38.565,179.802,5.366,148.994
C06860=1220.981,-63.961,-38.577,179.804,5.366,148.994
C06861=1220.976,-63.711,-38.589,179.807,5.366,148.993
C06862=1220.971,-63.461,-38.601,179.809,5.366,148.992
C06863=1220.966,-63.212,-38.613,179.812,5.367,148.992
C06864=1220.961,-62.962,-38.624,179.815,5.367,148.991
C06865=1220.955,-62.713,-38.636,179.817,5.367,148.990
C06866=1220.949,-62.463,-38.648,179.819,5.367,148.989
C06867=1220.945,-62.214,-38.660,179.821,5.367,148.989
C06868=1220.940,-61.964,-38.672,179.824,5.367,148.988
C06869=1220.934,-61.714,-38.684,179.826,5.367,148.987
C06870=1220.929,-61.464,-38.695,179.829,5.367,148.987
C06871=1220.924,-61.215,-38.707,179.831,5.368,148.986
C06872=1220.919,-60.965,-38.719,179.834,5.368,148.985
C06873=1220.913,-60.715,-38.731,179.836,5.368,148.984
C06874=1220.909,-60.466,-38.743,179.838,5.368,148.984
C06875=1220.904,-60.216,-38.755,179.840,5.368,148.983
C06876=1220.898,-59.966,-38.767,179.843,5.368,148.983
C06877=1220.894,-59.717,-38.778,179.845,5.369,148.982
C06878=1220.888,-59.467,-38.790,179.848,5.369,148.981
C06879=1220.883,-59.218,-38.803,179.850,5.369,148.980
C06880=1220.878,-58.968,-38.815,179.853,5.369,148.980
C06881=1220.873,-58.718,-38.826,179.855,5.369,148.979
C06882=1220.868,-58.469,-38.839,179.857,5.369,148.978
C06883=1220.862,-58.219,-38.850,179.860,5.369,148.978
C06884=1220.857,-57.969,-38.862,179.862,5.369,148.977
C06885=1220.853,-57.720,-38.874,179.865,5.370,148.976
C06886=1220.847,-57.470,-38.886,179.867,5.370,148.976
C06887=1220.842,-57.220,-38.898,179.870,5.370,148.975
C06888=1220.837,-56.971,-38.911,179.872,5.370,148.974
C06889=1220.831,-56.721,-38.923,179.874,5.370,148.973
C06890=1220.827,-56.472,-38.935,179.877,5.371,148.973
C06891=1220.821,-56.222,-38.946,179.879,5.370,148.972
C06892=1220.816,-55.972,-38.958,179.882,5.371,148.971
C06893=1220.811,-55.722,-38.971,179.884,5.370,148.971
C06894=1220.805,-55.473,-38.983,179.887,5.371,148.970
C06895=1220.801,-55.224,-38.995,179.889,5.371,148.969
C06896=1220.795,-54.974,-39.007,179.891,5.371,148.968
C06897=1220.791,-54.723,-39.019,179.894,5.372,148.968
C06898=1220.786,-54.474,-39.032,179.896,5.371,148.967
C06899=1220.780,-54.224,-39.043,179.899,5.372,148.966
C06900=1220.775,-53.974,-39.056,179.901,5.371,148.966
C06901=1220.770,-53.725,-39.067,179.903,5.372,148.965
C06902=1220.765,-53.475,-39.080,179.906,5.372,148.964
C06903=1220.760,-53.225,-39.092,179.908,5.372,148.964
C06904=1220.755,-52.976,-39.104,179.910,5.373,148.963
C06905=1220.749,-52.726,-39.116,179.912,5.372,148.962
C06906=1220.744,-52.477,-39.129,179.915,5.373,148.962
C06907=1220.739,-52.227,-39.141,179.918,5.373,148.961
C06908=1220.733,-51.978,-39.153,179.920,5.373,148.960
C06909=1220.729,-51.728,-39.165,179.923,5.373,148.960
C06910=1220.724,-51.478,-39.178,179.925,5.373,148.959
C06911=1220.719,-51.228,-39.190,179.927,5.374,148.958
C06912=1220.714,-50.979,-39.202,179.930,5.374,148.957
C06913=1220.708,-50.729,-39.214,179.932,5.374,148.957
C06914=1220.703,-50.480,-39.227,179.935,5.374,148.956
C06915=1220.698,-50.230,-39.239,179.937,5.374,148.955
C06916=1220.693,-49.980,-39.251,179.939,5.374,148.955
C06917=1220.687,-49.731,-39.264,179.942,5.375,148.954
C06918=1220.682,-49.481,-39.276,179.944,5.375,148.953
C06919=1220.678,-49.231,-39.289,179.947,5.375,148.953
C06920=1220.672,-48.961,-39.301,179.950,5.375,148.952
C06921=1220.667,-48.692,-39.315,179.952,5.375,148.951
C06922=1220.661,-48.421,-39.328,179.955,5.375,148.950
C06923=1220.655,-48.152,-39.342,179.957,5.376,148.949
C06924=1220.650,-47.903,-39.354,179.960,5.375,148.949
C06925=1220.644,-47.653,-39.366,179.962,5.376,148.948
C06926=1220.640,-47.403,-39.379,179.965,5.376,148.947
C06927=1220.634,-47.153,-39.391,179.967,5.376,148.947
C06928=1220.629,-46.903,-39.404,179.970,5.376,148.946
C06929=1220.624,-46.654,-39.416,179.972,5.376,148.945
C06930=1220.619,-46.404,-39.428,179.974,5.377,148.945
C06931=1220.614,-46.155,-39.441,179.977,5.377,148.944
C06932=1220.609,-45.905,-39.454,179.979,5.377,148.943
C06933=1220.604,-45.655,-39.466,179.982,5.377,148.942
C06934=1220.599,-45.406,-39.478,179.984,5.378,148.942
C06935=1220.593,-45.156,-39.491,179.986,5.378,148.941
C06936=1220.588,-44.907,-39.503,179.989,5.378,148.941
C06937=1220.584,-44.656,-39.516,179.991,5.378,148.940
C06938=1220.578,-44.407,-39.528,179.993,5.378,148.939
C06939=1220.573,-44.158,-39.541,179.996,5.379,148.938
C06940=1220.568,-43.908,-39.554,179.998,5.379,148.938
C06941=1220.563,-43.658,-39.565,-179.999,5.379,148.937
C06942=1220.558,-43.409,-39.578,-179.996,5.379,148.936
C06943=1220.553,-43.159,-39.591,-179.994,5.379,148.936
C06944=1220.548,-42.910,-39.604,-179.992,5.380,148.935
C06945=1220.543,-42.660,-39.615,-179.990,5.379,148.934
C06946=1220.537,-42.410,-39.629,-179.987,5.380,148.934
C06947=1220.532,-42.160,-39.642,-179.984,5.380,148.933
C06948=1220.527,-41.911,-39.654,-179.982,5.380,148.932
C06949=1220.522,-41.662,-39.667,-179.980,5.380,148.931
C06950=1220.516,-41.412,-39.679,-179.977,5.381,148.931
C06951=1220.512,-41.162,-39.692,-179.975,5.381,148.930
C06952=1220.507,-40.912,-39.704,-179.972,5.381,148.929
C06953=1220.502,-40.663,-39.717,-179.970,5.381,148.929
C06954=1220.496,-40.413,-39.730,-179.967,5.381,148.928
C06955=1220.491,-40.163,-39.743,-179.965,5.382,148.927
C06956=1220.486,-39.914,-39.756,-179.963,5.381,148.927
C06957=1220.481,-39.664,-39.768,-179.960,5.382,148.926
C06958=1220.476,-39.415,-39.780,-179.957,5.382,148.925
C06959=1220.471,-39.165,-39.793,-179.955,5.382,148.924
C06960=1220.466,-38.915,-39.806,-179.953,5.382,148.924
C06961=1220.460,-38.666,-39.819,-179.951,5.382,148.923
C06962=1220.455,-38.416,-39.831,-179.948,5.383,148.922
C06963=1220.450,-38.166,-39.844,-179.945,5.383,148.922
C06964=1220.445,-37.917,-39.857,-179.943,5.383,148.921
C06965=1220.440,-37.668,-39.870,-179.940,5.383,148.920
C06966=1220.434,-37.418,-39.883,-179.938,5.384,148.920
C06967=1220.430,-37.168,-39.896,-179.936,5.383,148.919
C06968=1220.424,-36.918,-39.908,-179.933,5.384,148.918
C06969=1220.419,-36.669,-39.920,-179.930,5.384,148.917
C06970=1220.415,-36.419,-39.933,-179.928,5.384,148.917
C06971=1220.409,-36.169,-39.946,-179.926,5.385,148.916
C06972=1220.404,-35.920,-39.959,-179.923,5.385,148.916
C06973=1220.399,-35.670,-39.972,-179.921,5.385,148.915
C06974=1220.394,-35.421,-39.985,-179.919,5.386,148.914
C06975=1220.388,-35.171,-39.998,-179.917,5.385,148.913
C06976=1220.384,-34.921,-40.011,-179.914,5.386,148.913
C06977=1220.379,-34.672,-40.023,-179.911,5.386,148.912
C06978=1220.374,-34.422,-40.036,-179.909,5.386,148.911
C06979=1220.368,-34.172,-40.050,-179.907,5.386,148.911
C06980=1220.363,-33.923,-40.062,-179.904,5.387,148.910
C06981=1220.358,-33.674,-40.075,-179.902,5.387,148.909
C06982=1220.353,-33.424,-40.089,-179.899,5.387,148.909
C06983=1220.348,-33.174,-40.102,-179.896,5.388,148.908
C06984=1220.343,-32.925,-40.114,-179.894,5.387,148.907
C06985=1220.338,-32.675,-40.127,-179.892,5.388,148.907
C06986=1220.332,-32.425,-40.140,-179.889,5.388,148.906
C06987=1220.327,-32.176,-40.153,-179.887,5.388,148.905
C06988=1220.323,-31.926,-40.166,-179.884,5.388,148.904
C06989=1220.317,-31.676,-40.179,-179.882,5.389,148.904
C06990=1220.312,-31.427,-40.192,-179.880,5.388,148.903
C06991=1220.307,-31.177,-40.205,-179.877,5.389,148.902
C06992=1220.302,-30.928,-40.219,-179.874,5.389,148.902
C06993=1220.297,-30.678,-40.232,-179.872,5.389,148.901
C06994=1220.292,-30.429,-40.244,-179.870,5.390,148.900
C06995=1220.286,-30.179,-40.257,-179.867,5.390,148.900
C06996=1220.282,-29.929,-40.270,-179.865,5.390,148.899
C06997=1220.277,-29.680,-40.283,-179.862,5.390,148.898
C06998=1220.272,-29.430,-40.297,-179.859,5.391,148.897
C06999=1220.266,-29.181,-40.310,-179.857,5.390,148.897
C07000=1220.261,-28.931,-40.323,-179.855,5.391,148.896
C07001=1220.256,-28.681,-40.336,-179.852,5.391,148.895
C07002=1220.251,-28.432,-40.349,-179.850,5.391,148.895
C07003=1220.246,-28.182,-40.363,-179.847,5.392,148.894
C07004=1220.241,-27.933,-40.375,-179.845,5.392,148.893
C07005=1220.236,-27.683,-40.388,-179.843,5.392,148.893
C07006=1220.230,-27.433,-40.402,-179.840,5.392,148.892
C07007=1220.225,-27.184,-40.414,-179.837,5.393,148.891
C07008=1220.220,-26.934,-40.429,-179.835,5.392,148.890
C07009=1220.215,-26.685,-40.441,-179.833,5.393,148.890
C07010=1220.210,-26.434,-40.455,-179.830,5.393,148.889
C07011=1220.205,-26.186,-40.468,-179.828,5.394,148.889
C07012=1220.201,-25.936,-40.481,-179.826,5.394,148.888
C07013=1220.195,-25.686,-40.494,-179.823,5.394,148.887
C07014=1220.190,-25.436,-40.507,-179.821,5.394,148.887
C07015=1220.185,-25.187,-40.521,-179.818,5.395,148.886
C07016=1220.180,-24.938,-40.534,-179.816,5.395,148.885
C07017=1220.174,-24.687,-40.547,-179.813,5.395,148.884
C07018=1220.170,-24.439,-40.561,-179.811,5.395,148.884
C07019=1220.164,-24.188,-40.574,-179.808,5.396,148.883
C07020=1220.159,-23.939,-40.587,-179.805,5.396,148.882
C07021=1220.154,-23.689,-40.601,-179.803,5.396,148.882
C07022=1220.149,-23.440,-40.614,-179.801,5.397,148.881
C07023=1220.144,-23.190,-40.627,-179.798,5.397,148.880
C07024=1220.139,-22.921,-40.642,-179.796,5.397,148.880
C07025=1220.133,-22.652,-40.656,-179.793,5.397,148.879
C07026=1220.127,-22.382,-40.670,-179.790,5.397,148.878
C07027=1220.123,-22.113,-40.685,-179.788,5.398,148.877
C07028=1220.117,-21.863,-40.698,-179.785,5.398,148.877
C07029=1220.113,-21.614,-40.712,-179.783,5.398,148.876
C07030=1220.107,-21.364,-40.725,-179.780,5.398,148.875
C07031=1220.101,-21.114,-40.738,-179.777,5.399,148.874
C07032=1220.097,-20.865,-40.752,-179.775,5.399,148.874
C07033=1220.091,-20.615,-40.765,-179.773,5.399,148.873
C07034=1220.087,-20.366,-40.779,-179.770,5.400,148.872
C07035=1220.081,-20.116,-40.792,-179.768,5.399,148.872
C07036=1220.076,-19.867,-40.806,-179.765,5.400,148.871
C07037=1220.071,-19.617,-40.819,-179.763,5.400,148.870
C07038=1220.066,-19.368,-40.833,-179.760,5.401,148.870
C07039=1220.061,-19.118,-40.846,-179.758,5.401,148.869
C07040=1220.056,-18.868,-40.860,-179.755,5.401,148.868
C07041=1220.051,-18.619,-40.873,-179.753,5.402,148.867
C07042=1220.046,-18.369,-40.887,-179.751,5.401,148.867
C07043=1220.040,-18.119,-40.900,-179.748,5.402,148.866
C07044=1220.036,-17.870,-40.914,-179.746,5.403,148.866
C07045=1220.030,-17.620,-40.927,-179.744,5.402,148.865
C07046=1220.026,-17.371,-40.941,-179.741,5.403,148.864
C07047=1220.021,-17.120,-40.954,-179.738,5.403,148.864
C07048=1220.015,-16.871,-40.968,-179.736,5.404,148.863
C07049=1220.011,-16.621,-40.981,-179.734,5.403,148.862
C07050=1220.005,-16.372,-40.995,-179.731,5.404,148.861
C07051=1220.000,-16.123,-41.009,-179.728,5.404,148.861
C07052=1219.995,-15.873,-41.022,-179.726,5.404,148.860
C07053=1219.990,-15.624,-41.036,-179.724,5.405,148.859
C07054=1219.985,-15.373,-41.050,-179.721,5.405,148.859
C07055=1219.980,-15.125,-41.063,-179.718,5.406,148.858
C07056=1219.975,-14.875,-41.078,-179.716,5.405,148.857
C07057=1219.969,-14.625,-41.091,-179.713,5.406,148.857
C07058=1219.965,-14.376,-41.104,-179.711,5.406,148.856
C07059=1219.960,-14.126,-41.118,-179.709,5.406,148.855
C07060=1219.954,-13.877,-41.132,-179.706,5.407,148.855
C07061=1219.949,-13.627,-41.146,-179.703,5.407,148.854
C07062=1219.945,-13.377,-41.159,-179.701,5.408,148.853
C07063=1219.939,-13.128,-41.173,-179.699,5.407,148.852
C07064=1219.934,-12.878,-41.187,-179.696,5.408,148.852
C07065=1219.930,-12.628,-41.200,-179.693,5.408,148.851
C07066=1219.924,-12.379,-41.214,-179.691,5.409,148.850
C07067=1219.919,-12.129,-41.228,-179.689,5.408,148.850
C07068=1219.914,-11.880,-41.242,-179.686,5.409,148.849
C07069=1219.909,-11.630,-41.255,-179.683,5.409,148.848
C07070=1219.904,-11.381,-41.270,-179.681,5.409,148.848
C07071=1219.898,-11.132,-41.284,-179.679,5.410,148.847
C07072=1219.894,-10.882,-41.298,-179.676,5.410,148.846
C07073=1219.889,-10.632,-41.311,-179.674,5.411,148.846
C07074=1219.883,-10.383,-41.325,-179.672,5.411,148.845
C07075=1219.879,-10.133,-41.339,-179.669,5.411,148.844
C07076=1219.874,-9.883,-41.353,-179.666,5.412,148.844
C07077=1219.868,-9.633,-41.367,-179.664,5.412,148.843
C07078=1219.863,-9.384,-41.380,-179.662,5.412,148.842
C07079=1219.859,-9.135,-41.394,-179.659,5.412,148.842
C07080=1219.854,-8.885,-41.409,-179.656,5.413,148.841
C07081=1219.848,-8.636,-41.423,-179.654,5.413,148.840
C07082=1219.843,-8.386,-41.436,-179.652,5.413,148.840
C07083=1219.839,-8.136,-41.450,-179.649,5.414,148.839
C07084=1219.833,-7.887,-41.464,-179.646,5.414,148.838
C07085=1219.828,-7.638,-41.478,-179.644,5.414,148.837
C07086=1219.823,-7.388,-41.492,-179.642,5.414,148.837
C07087=1219.818,-7.138,-41.507,-179.639,5.415,148.836
C07088=1219.812,-6.889,-41.520,-179.636,5.415,148.835
C07089=1219.808,-6.639,-41.533,-179.634,5.415,148.835
C07090=1219.803,-6.389,-41.548,-179.632,5.416,148.834
C07091=1219.798,-6.140,-41.562,-179.629,5.416,148.833
C07092=1219.793,-5.891,-41.576,-179.626,5.417,148.833
C07093=1219.788,-5.641,-41.590,-179.624,5.416,148.832
C07094=1219.783,-5.391,-41.604,-179.621,5.417,148.831
C07095=1219.777,-5.142,-41.618,-179.619,5.417,148.831
C07096=1219.772,-4.893,-41.633,-179.616,5.418,148.830
C07097=1219.767,-4.643,-41.647,-179.614,5.418,148.829
C07098=1219.763,-4.393,-41.660,-179.612,5.418,148.829
C07099=1219.758,-4.143,-41.674,-179.609,5.419,148.828
C07100=1219.752,-3.894,-41.688,-179.607,5.419,148.827
C07101=1219.747,-3.644,-41.702,-179.604,5.420,148.827
C07102=1219.742,-3.395,-41.717,-179.602,5.420,148.826
C07103=1219.737,-3.145,-41.731,-179.599,5.420,148.825
C07104=1219.732,-2.896,-41.745,-179.597,5.421,148.825
C07105=1219.727,-2.646,-41.759,-179.594,5.421,148.824
C07106=1219.722,-2.397,-41.773,-179.592,5.421,148.823
C07107=1219.717,-2.147,-41.788,-179.589,5.421,148.822
C07108=1219.712,-1.897,-41.802,-179.587,5.422,148.822
C07109=1219.706,-1.648,-41.816,-179.584,5.422,148.821
C07110=1219.701,-1.398,-41.830,-179.582,5.422,148.820
C07111=1219.696,-1.149,-41.844,-179.579,5.423,148.820
C07112=1219.691,-0.899,-41.859,-179.577,5.423,148.819
C07113=1219.687,-0.650,-41.874,-179.574,5.424,148.818
C07114=1219.681,-0.401,-41.888,-179.572,5.423,148.818
C07115=1219.676,-0.151,-41.902,-179.569,5.424,148.817
C07116=1219.671,0.099,-41.916,-179.566,5.424,148.816
C07117=1219.666,0.348,-41.930,-179.564,5.425,148.816
C07118=1219.661,0.598,-41.945,-179.561,5.425,148.815
C07119=1219.657,0.848,-41.959,-179.560,5.426,148.814
C07120=1219.651,1.097,-41.973,-179.557,5.426,148.814
C07121=1219.646,1.346,-41.987,-179.554,5.427,148.813
C07122=1219.641,1.596,-42.001,-179.552,5.427,148.812
C07123=1219.636,1.845,-42.016,-179.550,5.427,148.812
C07124=1219.631,2.095,-42.031,-179.547,5.427,148.811
C07125=1219.626,2.345,-42.045,-179.544,5.428,148.810
C07126=1219.621,2.594,-42.059,-179.542,5.428,148.810
C07127=1219.616,2.843,-42.073,-179.539,5.429,148.809
C07128=1219.611,3.112,-42.089,-179.537,5.429,148.808
C07129=1219.605,3.382,-42.104,-179.534,5.429,148.808
C07130=1219.600,3.651,-42.120,-179.531,5.429,148.807
C07131=1219.594,3.919,-42.136,-179.528,5.430,148.806
C07132=1219.589,4.169,-42.150,-179.526,5.430,148.805
C07133=1219.585,4.419,-42.164,-179.523,5.431,148.805
C07134=1219.580,4.669,-42.179,-179.520,5.431,148.804
C07135=1219.574,4.917,-42.193,-179.519,5.431,148.803
C07136=1219.569,5.167,-42.208,-179.516,5.432,148.803
C07137=1219.564,5.417,-42.222,-179.514,5.432,148.802
C07138=1219.559,5.666,-42.237,-179.511,5.433,148.801
C07139=1219.554,5.916,-42.252,-179.508,5.433,148.801
C07140=1219.549,6.165,-42.266,-179.506,5.433,148.800
C07141=1219.544,6.415,-42.280,-179.504,5.434,148.799
C07142=1219.540,6.664,-42.295,-179.501,5.434,148.799
C07143=1219.534,6.914,-42.310,-179.498,5.435,148.798
C07144=1219.529,7.164,-42.324,-179.496,5.435,148.797
C07145=1219.524,7.413,-42.339,-179.494,5.435,148.797
C07146=1219.519,7.663,-42.354,-179.491,5.435,148.796
C07147=1219.514,7.912,-42.368,-179.488,5.436,148.795
C07148=1219.509,8.161,-42.382,-179.486,5.437,148.795
C07149=1219.503,8.411,-42.398,-179.483,5.437,148.794
C07150=1219.498,8.660,-42.412,-179.481,5.437,148.793
C07151=1219.493,8.910,-42.426,-179.479,5.438,148.793
C07152=1219.489,9.159,-42.441,-179.476,5.438,148.792
C07153=1219.484,9.409,-42.455,-179.473,5.439,148.791
C07154=1219.478,9.658,-42.471,-179.471,5.439,148.791
C07155=1219.473,9.908,-42.485,-179.469,5.439,148.790
C07156=1219.469,10.158,-42.499,-179.466,5.439,148.789
C07157=1219.464,10.407,-42.514,-179.463,5.440,148.789
C07158=1219.458,10.657,-42.529,-179.461,5.440,148.788
C07159=1219.454,10.906,-42.544,-179.458,5.441,148.787
C07160=1219.449,11.156,-42.559,-179.455,5.442,148.787
C07161=1219.444,11.405,-42.574,-179.453,5.441,148.786
C07162=1219.438,11.655,-42.588,-179.451,5.442,148.785
C07163=1219.433,11.904,-42.603,-179.448,5.442,148.784
C07164=1219.429,12.154,-42.618,-179.445,5.443,148.784
C07165=1219.424,12.403,-42.632,-179.443,5.443,148.783
C07166=1219.418,12.653,-42.648,-179.441,5.443,148.783
C07167=1219.413,12.902,-42.662,-179.439,5.444,148.782
C07168=1219.409,13.151,-42.677,-179.436,5.444,148.781
C07169=1219.403,13.401,-42.692,-179.433,5.445,148.781
C07170=1219.398,13.651,-42.707,-179.431,5.446,148.780
C07171=1219.393,13.900,-42.721,-179.428,5.446,148.779
C07172=1219.388,14.150,-42.737,-179.426,5.446,148.779
C07173=1219.383,14.399,-42.751,-179.423,5.446,148.778
C07174=1219.378,14.648,-42.766,-179.421,5.447,148.777
C07175=1219.373,14.899,-42.781,-179.418,5.447,148.776
C07176=1219.368,15.148,-42.796,-179.415,5.448,148.776
C07177=1219.363,15.397,-42.811,-179.413,5.448,148.775
C07178=1219.358,15.647,-42.826,-179.411,5.448,148.774
C07179=1219.353,15.896,-42.841,-179.408,5.449,148.774
C07180=1219.349,16.146,-42.855,-179.406,5.450,148.773
C07181=1219.343,16.396,-42.871,-179.403,5.450,148.773
C07182=1219.339,16.645,-42.886,-179.400,5.451,148.772
C07183=1219.333,16.895,-42.901,-179.398,5.451,148.771
C07184=1219.328,17.144,-42.916,-179.396,5.451,148.771
C07185=1219.323,17.394,-42.930,-179.393,5.451,148.770
C07186=1219.318,17.643,-42.946,-179.390,5.452,148.769
C07187=1219.313,17.892,-42.961,-179.388,5.452,148.769
C07188=1219.308,18.142,-42.975,-179.385,5.453,148.768
C07189=1219.303,18.391,-42.990,-179.382,5.453,148.767
C07190=1219.298,18.640,-43.005,-179.380,5.454,148.766
C07191=1219.293,18.890,-43.020,-179.378,5.454,148.766
C07192=1219.289,19.140,-43.036,-179.376,5.455,148.765
C07193=1219.283,19.389,-43.051,-179.373,5.455,148.765
C07194=1219.278,19.639,-43.066,-179.370,5.456,148.764
C07195=1219.273,19.889,-43.081,-179.368,5.456,148.763
C07196=1219.268,20.138,-43.096,-179.365,5.457,148.763
C07197=1219.263,20.387,-43.112,-179.363,5.456,148.762
C07198=1219.258,20.637,-43.126,-179.360,5.457,148.761
C07199=1219.253,20.886,-43.141,-179.358,5.458,148.761
C07200=1219.248,21.136,-43.157,-179.355,5.458,148.760
C07201=1219.244,21.385,-43.172,-179.352,5.459,148.759
C07202=1219.238,21.635,-43.187,-179.350,5.459,148.759
C07203=1219.233,21.884,-43.202,-179.348,5.460,148.758
C07204=1219.228,22.134,-43.217,-179.345,5.460,148.757
C07205=1219.223,22.383,-43.232,-179.343,5.460,148.757
C07206=1219.218,22.633,-43.247,-179.340,5.461,148.756
C07207=1219.213,22.883,-43.263,-179.338,5.461,148.755
C07208=1219.208,23.132,-43.278,-179.335,5.462,148.755
C07209=1219.203,23.381,-43.294,-179.332,5.462,148.754
C07210=1219.198,23.630,-43.309,-179.330,5.463,148.753
C07211=1219.193,23.880,-43.324,-179.327,5.463,148.753
C07212=1219.188,24.129,-43.339,-179.325,5.463,148.752
C07213=1219.183,24.380,-43.355,-179.323,5.464,148.751
C07214=1219.179,24.629,-43.370,-179.320,5.465,148.751
C07215=1219.173,24.878,-43.385,-179.317,5.465,148.750
C07216=1219.168,25.127,-43.400,-179.315,5.466,148.749
C07217=1219.163,25.377,-43.416,-179.312,5.466,148.749
C07218=1219.158,25.627,-43.432,-179.309,5.467,148.748
C07219=1219.154,25.876,-43.447,-179.307,5.467,148.747
C07220=1219.148,26.125,-43.462,-179.305,5.467,148.747
C07221=1219.143,26.375,-43.477,-179.302,5.468,148.746
C07222=1219.138,26.624,-43.492,-179.299,5.468,148.745
C07223=1219.133,26.874,-43.508,-179.297,5.469,148.745
C07224=1219.128,27.123,-43.523,-179.295,5.470,148.744
C07225=1219.123,27.373,-43.539,-179.292,5.470,148.744
C07226=1219.118,27.622,-43.554,-179.289,5.471,148.743
C07227=1219.114,27.872,-43.570,-179.287,5.471,148.742
C07228=1219.108,28.121,-43.585,-179.285,5.471,148.742
C07229=1219.104,28.371,-43.600,-179.282,5.471,148.741
C07230=1219.098,28.620,-43.616,-179.279,5.472,148.740
C07231=1219.093,28.870,-43.632,-179.277,5.473,148.739
C07232=1219.089,29.138,-43.648,-179.274,5.473,148.739
C07233=1219.083,29.407,-43.664,-179.271,5.474,148.738
C07234=1219.077,29.676,-43.681,-179.269,5.474,148.737
C07235=1219.072,29.944,-43.698,-179.266,5.475,148.737
C07236=1219.067,30.193,-43.713,-179.264,5.475,148.736
C07237=1219.062,30.444,-43.729,-179.261,5.476,148.735
C07238=1219.057,30.693,-43.745,-179.258,5.476,148.735
C07239=1219.052,30.942,-43.760,-179.256,5.477,148.734
C07240=1219.047,31.191,-43.776,-179.253,5.478,148.734
C07241=1219.042,31.442,-43.792,-179.251,5.478,148.733
C07242=1219.037,31.691,-43.807,-179.248,5.479,148.732
C07243=1219.032,31.939,-43.823,-179.246,5.479,148.732
C07244=1219.028,32.189,-43.839,-179.243,5.479,148.731
C07245=1219.022,32.439,-43.854,-179.241,5.480,148.730
C07246=1219.017,32.688,-43.870,-179.238,5.480,148.730
C07247=1219.013,32.938,-43.885,-179.236,5.481,148.729
C07248=1219.007,33.187,-43.901,-179.233,5.481,148.728
C07249=1219.002,33.437,-43.917,-179.231,5.482,148.728
C07250=1218.997,33.686,-43.932,-179.228,5.483,148.727
C07251=1218.993,33.935,-43.948,-179.225,5.483,148.726
C07252=1218.987,34.185,-43.964,-179.223,5.484,148.726
C07253=1218.982,34.434,-43.979,-179.220,5.484,148.725
C07254=1218.977,34.684,-43.995,-179.217,5.485,148.724
C07255=1218.973,34.933,-44.010,-179.215,5.485,148.724
C07256=1218.967,35.182,-44.027,-179.213,5.485,148.723
C07257=1218.963,35.432,-44.043,-179.211,5.486,148.723
C07258=1218.957,35.682,-44.058,-179.208,5.487,148.722
C07259=1218.953,35.932,-44.074,-179.205,5.487,148.721
C07260=1218.947,36.181,-44.090,-179.203,5.488,148.721
C07261=1218.943,36.430,-44.105,-179.200,5.488,148.720
C07262=1218.938,36.680,-44.121,-179.197,5.489,148.719
C07263=1218.933,36.929,-44.137,-179.195,5.489,148.719
C07264=1218.928,37.178,-44.153,-179.193,5.490,148.718
C07265=1218.923,37.428,-44.169,-179.190,5.491,148.717
C07266=1218.917,37.678,-44.185,-179.187,5.491,148.717
C07267=1218.913,37.928,-44.201,-179.185,5.492,148.716
C07268=1218.908,38.176,-44.216,-179.182,5.492,148.715
C07269=1218.903,38.425,-44.232,-179.180,5.492,148.715
C07270=1218.898,38.676,-44.248,-179.177,5.493,148.714
C07271=1218.893,38.924,-44.264,-179.175,5.493,148.713
C07272=1218.888,39.174,-44.280,-179.173,5.494,148.713
C07273=1218.883,39.424,-44.296,-179.170,5.495,148.712
C07274=1218.878,39.673,-44.312,-179.167,5.495,148.712
C07275=1218.873,39.923,-44.328,-179.165,5.496,148.711
C07276=1218.868,40.172,-44.344,-179.162,5.496,148.710
C07277=1218.863,40.422,-44.360,-179.159,5.497,148.710
C07278=1218.858,40.671,-44.376,-179.157,5.497,148.709
C07279=1218.853,40.920,-44.392,-179.155,5.498,148.708
C07280=1218.849,41.170,-44.408,-179.152,5.499,148.708
C07281=1218.843,41.418,-44.424,-179.149,5.499,148.707
C07282=1218.839,41.669,-44.440,-179.147,5.500,148.706
C07283=1218.833,41.918,-44.455,-179.144,5.501,148.706
C07284=1218.829,42.167,-44.472,-179.141,5.501,148.705
C07285=1218.823,42.417,-44.488,-179.139,5.502,148.704
C07286=1218.819,42.666,-44.504,-179.137,5.503,148.704
C07287=1218.814,42.916,-44.520,-179.135,5.502,148.703
C07288=1218.809,43.164,-44.536,-179.132,5.503,148.703
C07289=1218.804,43.415,-44.552,-179.129,5.503,148.702
C07290=1218.799,43.663,-44.569,-179.127,5.504,148.701
C07291=1218.794,43.913,-44.584,-179.124,5.505,148.701
C07292=1218.789,44.162,-44.601,-179.122,5.505,148.700
C07293=1218.784,44.412,-44.617,-179.119,5.506,148.699
C07294=1218.779,44.661,-44.633,-179.117,5.507,148.699
C07295=1218.774,44.911,-44.649,-179.114,5.507,148.698
C07296=1218.769,45.160,-44.665,-179.111,5.508,148.697
C07297=1218.764,45.410,-44.681,-179.109,5.508,148.697
C07298=1218.759,45.659,-44.698,-179.106,5.509,148.696
C07299=1218.754,45.909,-44.714,-179.104,5.510,148.696
C07300=1218.749,46.158,-44.730,-179.101,5.510,148.695
C07301=1218.744,46.408,-44.747,-179.099,5.511,148.694
C07302=1218.739,46.657,-44.763,-179.096,5.511,148.694
C07303=1218.734,46.906,-44.779,-179.093,5.512,148.693
C07304=1218.729,47.156,-44.795,-179.091,5.512,148.692
C07305=1218.724,47.405,-44.812,-179.089,5.513,148.692
C07306=1218.720,47.655,-44.828,-179.086,5.514,148.691
C07307=1218.714,47.904,-44.844,-179.083,5.514,148.691
C07308=1218.710,48.154,-44.860,-179.081,5.515,148.690
C07309=1218.705,48.403,-44.877,-179.078,5.516,148.689
C07310=1218.700,48.653,-44.893,-179.075,5.516,148.689
